LIN {X 0,Y 573.093,Z 692.429,A -85,B 0,C 180,E1 -2257.751,E2 -2257.751} C_VEL
LIN {X 0,Y 573.135,Z 684.656,A -85,B 0,C 180,E1 -2259.172,E2 -2259.172} C_VEL
LIN {X 0,Y 573.27,Z 676.378,A -85,B 0,C 180,E1 -2260.417,E2 -2260.417} C_VEL
LIN {X 0,Y 573.384,Z 666.402,A -85,B 0,C 180,E1 -2261.667,E2 -2261.667} C_VEL
LIN {X 0,Y 573.566,Z 656.201,A -85,B 0,C 180,E1 -2262.741,E2 -2262.741} C_VEL
LIN {X 0,Y 573.742,Z 644.034,A -85,B 0,C 180,E1 -2263.818,E2 -2263.818} C_VEL
LIN {X 0,Y 573.958,Z 630.922,A -85,B 0,C 180,E1 -2264.78,E2 -2264.78} C_VEL
LIN {X 0,Y 574.109,Z 618.538,A -85,B 0,C 180,E1 -2265.531,E2 -2265.531} C_VEL
LIN {X 0,Y 574.343,Z 603.86,A -85,B 0,C 180,E1 -2266.254,E2 -2266.254} C_VEL
LIN {X 0,Y 574.537,Z 589.652,A -85,B 0,C 180,E1 -2266.796,E2 -2266.796} C_VEL
LIN {X 0,Y 574.697,Z 574.641,A -85,B 0,C 180,E1 -2267.221,E2 -2267.221} C_VEL
LIN {X 0,Y 574.75,Z 559.765,A -85,B 0,C 180,E1 -2267.501,E2 -2267.501} C_VEL
LIN {X 0,Y 575.189,Z 405.134,A -85,B 0,C 180,E1 -2269.487,E2 -2269.487} C_VEL
LIN {X 0,Y 574.004,Z 398.788,A -85,B 0,C 180,E1 -2269.625,E2 -2269.625} C_VEL
LIN {X 0,Y 574.346,Z 373.403,A -85,B 0,C 180,E1 -2272.67,E2 -2272.67} C_VEL
LIN {X 0,Y 574.669,Z 351.554,A -85,B 0,C 180,E1 -2275.342,E2 -2275.342} C_VEL
LIN {X 0,Y 573.967,Z 346.839,A -85,B 0,C 180,E1 -2275.959,E2 -2275.959} C_VEL
LIN {X 0,Y 573.219,Z 343.711,A -85,B 0,C 180,E1 -2276.413,E2 -2276.413} C_VEL
LIN {X 0,Y 573.236,Z 343.702,A -85,B 0,C 180,E1 -2279.366,E2 -2279.366} C_VEL
LIN {X 0,Y 573.239,Z 343.709,A -85,B 0,C 180,E1 -2282.226,E2 -2282.226} C_VEL
LIN {X 0,Y 573.211,Z 343.705,A -85,B 0,C 180,E1 -2284.768,E2 -2284.768} C_VEL
LIN {X 0,Y 573.211,Z 343.707,A -85,B 0,C 180,E1 -2287.808,E2 -2287.808} C_VEL
LIN {X 0,Y 573.235,Z 343.704,A -85,B 0,C 180,E1 -2290.524,E2 -2290.524} C_VEL
LIN {X 0,Y 573.189,Z 343.705,A -85,B 0,C 180,E1 -2293.362,E2 -2293.362} C_VEL
LIN {X 0,Y 573.193,Z 343.712,A -85,B 0,C 180,E1 -2296.334,E2 -2296.334} C_VEL
LIN {X 0,Y 573.191,Z 343.709,A -85,B 0,C 180,E1 -2298.54,E2 -2298.54} C_VEL
LIN {X 0,Y 573.219,Z 343.701,A -85,B 0,C 180,E1 -2301.297,E2 -2301.297} C_VEL
LIN {X 0,Y 573.172,Z 343.715,A -85,B 0,C 180,E1 -2304.021,E2 -2304.021} C_VEL
LIN {X 0,Y 573.236,Z 343.703,A -85,B 0,C 180,E1 -2306.516,E2 -2306.516} C_VEL
LIN {X 0,Y 573.208,Z 343.703,A -85,B 0,C 180,E1 -2309.118,E2 -2309.118} C_VEL
LIN {X 0,Y 573.188,Z 343.713,A -85,B 0,C 180,E1 -2311.98,E2 -2311.98} C_VEL
LIN {X 0,Y 573.213,Z 343.705,A -85,B 0,C 180,E1 -2314.588,E2 -2314.588} C_VEL
LIN {X 0,Y 573.201,Z 343.707,A -85,B 0,C 180,E1 -2317.661,E2 -2317.661} C_VEL
LIN {X 0,Y 573.253,Z 343.698,A -85,B 0,C 180,E1 -2320.731,E2 -2320.731} C_VEL
LIN {X 0,Y 573.191,Z 343.708,A -85,B 0,C 180,E1 -2323.62,E2 -2323.62} C_VEL
LIN {X 0,Y 573.239,Z 343.705,A -85,B 0,C 180,E1 -2325.806,E2 -2325.806} C_VEL
LIN {X 0,Y 573.247,Z 343.699,A -85,B 0,C 180,E1 -2328.745,E2 -2328.745} C_VEL
LIN {X 0,Y 573.228,Z 343.703,A -85,B 0,C 180,E1 -2331.54,E2 -2331.54} C_VEL
LIN {X 0,Y 573.259,Z 343.701,A -85,B 0,C 180,E1 -2334.372,E2 -2334.372} C_VEL
LIN {X 0,Y 573.297,Z 343.7,A -85,B 0,C 180,E1 -2337.893,E2 -2337.893} C_VEL
LIN {X 0,Y 573.303,Z 343.701,A -85,B 0,C 180,E1 -2340,E2 -2340} C_VEL
LIN {X 0,Y 573.255,Z 343.697,A -85,B 0,C 180,E1 -2342.811,E2 -2342.811} C_VEL
LIN {X 0,Y 573.252,Z 343.702,A -85,B 0,C 180,E1 -2345.629,E2 -2345.629} C_VEL
LIN {X 0,Y 573.228,Z 343.703,A -85,B 0,C 180,E1 -2348.461,E2 -2348.461} C_VEL
LIN {X 0,Y 573.219,Z 343.703,A -85,B 0,C 180,E1 -2351.313,E2 -2351.313} C_VEL
LIN {X 0,Y 573.255,Z 343.7,A -85,B 0,C 180,E1 -2354.42,E2 -2354.42} C_VEL
LIN {X 0,Y 573.179,Z 343.707,A -85,B 0,C 180,E1 -2357.114,E2 -2357.114} C_VEL
LIN {X 0,Y 573.25,Z 343.699,A -85,B 0,C 180,E1 -2359.331,E2 -2359.331} C_VEL
LIN {X 0,Y 573.202,Z 343.707,A -85,B 0,C 180,E1 -2362.339,E2 -2362.339} C_VEL
LIN {X 0,Y 573.189,Z 343.708,A -85,B 0,C 180,E1 -2364.354,E2 -2364.354} C_VEL
LIN {X 0,Y 572.546,Z 343.788,A -85,B 0,C 180,E1 -2364.94,E2 -2364.94} C_VEL
LIN {X 0,Y 569.708,Z 344.149,A -85,B 0,C 180,E1 -2365.892,E2 -2365.892} C_VEL
LIN {X 0,Y 567.287,Z 344.447,A -85,B 0,C 180,E1 -2366.658,E2 -2366.658} C_VEL
LIN {X 0,Y 566.232,Z 344.574,A -85,B 0,C 180,E1 -2367.249,E2 -2367.249} C_VEL
LIN {X 0,Y 566.139,Z 344.585,A -85,B 0,C 180,E1 -2367.449,E2 -2367.449} C_VEL
LIN {X 0,Y 566.154,Z 344.582,A -85,B 0,C 180,E1 -2370.595,E2 -2370.595} C_VEL
LIN {X 0,Y 566.196,Z 344.577,A -85,B 0,C 180,E1 -2373.104,E2 -2373.104} C_VEL
LIN {X 0,Y 566.128,Z 344.592,A -85,B 0,C 180,E1 -2375.695,E2 -2375.695} C_VEL
LIN {X 0,Y 566.191,Z 344.578,A -85,B 0,C 180,E1 -2378.558,E2 -2378.558} C_VEL
LIN {X 0,Y 566.145,Z 344.583,A -85,B 0,C 180,E1 -2381.143,E2 -2381.143} C_VEL
LIN {X 0,Y 566.148,Z 344.589,A -85,B 0,C 180,E1 -2384.041,E2 -2384.041} C_VEL
LIN {X 0,Y 566.178,Z 344.579,A -85,B 0,C 180,E1 -2387.086,E2 -2387.086} C_VEL
LIN {X 0,Y 566.201,Z 344.578,A -85,B 0,C 180,E1 -2390.316,E2 -2390.316} C_VEL
LIN {X 0,Y 566.167,Z 344.584,A -85,B 0,C 180,E1 -2393.429,E2 -2393.429} C_VEL
LIN {X 0,Y 566.191,Z 344.58,A -85,B 0,C 180,E1 -2396.27,E2 -2396.27} C_VEL
LIN {X 0,Y 566.182,Z 344.578,A -85,B 0,C 180,E1 -2398.926,E2 -2398.926} C_VEL
LIN {X 0,Y 566.147,Z 344.591,A -85,B 0,C 180,E1 -2401.855,E2 -2401.855} C_VEL
LIN {X 0,Y 566.184,Z 344.58,A -85,B 0,C 180,E1 -2404.251,E2 -2404.251} C_VEL
LIN {X 0,Y 566.164,Z 344.58,A -85,B 0,C 180,E1 -2406.722,E2 -2406.722} C_VEL
LIN {X 0,Y 566.2,Z 344.585,A -85,B 0,C 180,E1 -2409.664,E2 -2409.664} C_VEL
LIN {X 0,Y 566.17,Z 344.586,A -85,B 0,C 180,E1 -2411.922,E2 -2411.922} C_VEL
LIN {X 0,Y 566.185,Z 344.578,A -85,B 0,C 180,E1 -2414.891,E2 -2414.891} C_VEL
LIN {X 0,Y 566.214,Z 344.582,A -85,B 0,C 180,E1 -2417.82,E2 -2417.82} C_VEL
LIN {X 0,Y 566.164,Z 344.585,A -85,B 0,C 180,E1 -2419.993,E2 -2419.993} C_VEL
LIN {X 0,Y 566.192,Z 344.58,A -85,B 0,C 180,E1 -2422.153,E2 -2422.153} C_VEL
LIN {X 0,Y 566.261,Z 344.569,A -85,B 0,C 180,E1 -2425.017,E2 -2425.017} C_VEL
LIN {X 0,Y 566.281,Z 344.572,A -85,B 0,C 180,E1 -2427.867,E2 -2427.867} C_VEL
LIN {X 0,Y 566.288,Z 344.569,A -85,B 0,C 180,E1 -2430.001,E2 -2430.001} C_VEL
LIN {X 0,Y 566.248,Z 344.57,A -85,B 0,C 180,E1 -2432.847,E2 -2432.847} C_VEL
LIN {X 0,Y 566.247,Z 344.579,A -85,B 0,C 180,E1 -2435.699,E2 -2435.699} C_VEL
LIN {X 0,Y 566.201,Z 344.576,A -85,B 0,C 180,E1 -2438.567,E2 -2438.567} C_VEL
LIN {X 0,Y 566.245,Z 344.578,A -85,B 0,C 180,E1 -2441.455,E2 -2441.455} C_VEL
LIN {X 0,Y 566.224,Z 344.573,A -85,B 0,C 180,E1 -2444.501,E2 -2444.501} C_VEL
LIN {X 0,Y 566.159,Z 344.587,A -85,B 0,C 180,E1 -2447.334,E2 -2447.334} C_VEL
LIN {X 0,Y 566.205,Z 344.586,A -85,B 0,C 180,E1 -2449.582,E2 -2449.582} C_VEL
LIN {X 0,Y 566.191,Z 344.582,A -85,B 0,C 180,E1 -2451.864,E2 -2451.864} C_VEL
LIN {X 0,Y 566.185,Z 344.58,A -85,B 0,C 180,E1 -2455.022,E2 -2455.022} C_VEL
LIN {X 0,Y 566.172,Z 344.586,A -85,B 0,C 180,E1 -2457.342,E2 -2457.342} C_VEL
LIN {X 0,Y 566.177,Z 344.585,A -85,B 0,C 180,E1 -2459.771,E2 -2459.771} C_VEL
LIN {X 0,Y 566.205,Z 344.575,A -85,B 0,C 180,E1 -2462.429,E2 -2462.429} C_VEL
LIN {X 0,Y 566.174,Z 344.581,A -85,B 0,C 180,E1 -2464.988,E2 -2464.988} C_VEL
LIN {X 0,Y 566.197,Z 344.587,A -85,B 0,C 180,E1 -2467.462,E2 -2467.462} C_VEL
LIN {X 0,Y 566.212,Z 344.577,A -85,B 0,C 180,E1 -2470.199,E2 -2470.199} C_VEL
LIN {X 0,Y 566.197,Z 344.581,A -85,B 0,C 180,E1 -2473.055,E2 -2473.055} C_VEL
LIN {X 0,Y 566.164,Z 344.587,A -85,B 0,C 180,E1 -2476.053,E2 -2476.053} C_VEL
LIN {X 0,Y 566.24,Z 344.709,A -85,B 0,C 180,E1 -2477.589,E2 -2477.589} C_VEL
LIN {X 0,Y 567.165,Z 350.607,A -85,B 0,C 180,E1 -2478.475,E2 -2478.475} C_VEL
LIN {X 0,Y 566.907,Z 369.86,A -85,B 0,C 180,E1 -2481.181,E2 -2481.181} C_VEL
LIN {X 0,Y 568.471,Z 377.974,A -85,B 0,C 180,E1 -2481.356,E2 -2481.356} C_VEL
LIN {X 0,Y 567.987,Z 535.046,A -85,B 0,C 180,E1 -2483.412,E2 -2483.412} C_VEL
LIN {X 0,Y 567.798,Z 550.912,A -85,B 0,C 180,E1 -2483.769,E2 -2483.769} C_VEL
LIN {X 0,Y 567.621,Z 565.523,A -85,B 0,C 180,E1 -2484.25,E2 -2484.25} C_VEL
LIN {X 0,Y 567.413,Z 579.054,A -85,B 0,C 180,E1 -2484.834,E2 -2484.834} C_VEL
LIN {X 0,Y 567.18,Z 590.968,A -85,B 0,C 180,E1 -2485.466,E2 -2485.466} C_VEL
LIN {X 0,Y 566.958,Z 603.145,A -85,B 0,C 180,E1 -2486.234,E2 -2486.234} C_VEL
LIN {X 0,Y 566.694,Z 616.436,A -85,B 0,C 180,E1 -2487.254,E2 -2487.254} C_VEL
LIN {X 0,Y 566.474,Z 628.594,A -85,B 0,C 180,E1 -2488.387,E2 -2488.387} C_VEL
LIN {X 0,Y 566.315,Z 639.636,A -85,B 0,C 180,E1 -2489.621,E2 -2489.621} C_VEL
LIN {X 0,Y 566.174,Z 648.775,A -85,B 0,C 180,E1 -2490.842,E2 -2490.842} C_VEL
LIN {X 0,Y 566.081,Z 656.346,A -85,B 0,C 180,E1 -2492.051,E2 -2492.051} C_VEL
LIN {X 0,Y 565.985,Z 663.625,A -85,B 0,C 180,E1 -2493.447,E2 -2493.447} C_VEL
LIN {X 0,Y 565.937,Z 668.628,A -85,B 0,C 180,E1 -2494.632,E2 -2494.632} C_VEL
LIN {X 0,Y 565.902,Z 672.635,A -85,B 0,C 180,E1 -2495.806,E2 -2495.806} C_VEL
LIN {X 0,Y 565.858,Z 676.627,A -85,B 0,C 180,E1 -2497.355,E2 -2497.355} C_VEL
LIN {X 0,Y 565.879,Z 679.184,A -85,B 0,C 180,E1 -2498.889,E2 -2498.889} C_VEL
LIN {X 0,Y 565.828,Z 680.353,A -85,B 0,C 180,E1 -2500.405,E2 -2500.405} C_VEL
LIN {X 0,Y 565.834,Z 680.288,A -85,B 0,C 180,E1 -2501.909,E2 -2501.909} C_VEL
LIN {X 0,Y 565.849,Z 678.914,A -85,B 0,C 180,E1 -2503.401,E2 -2503.401} C_VEL
LIN {X 0,Y 565.836,Z 676.338,A -85,B 0,C 180,E1 -2504.88,E2 -2504.88} C_VEL
LIN {X 0,Y 565.906,Z 672.428,A -85,B 0,C 180,E1 -2506.351,E2 -2506.351} C_VEL
LIN {X 0,Y 565.95,Z 667.235,A -85,B 0,C 180,E1 -2507.813,E2 -2507.813} C_VEL
LIN {X 0,Y 566.022,Z 660.559,A -85,B 0,C 180,E1 -2509.266,E2 -2509.266} C_VEL
LIN {X 0,Y 566.104,Z 652.29,A -85,B 0,C 180,E1 -2510.712,E2 -2510.712} C_VEL
LIN {X 0,Y 566.277,Z 643.544,A -85,B 0,C 180,E1 -2511.974,E2 -2511.974} C_VEL
LIN {X 0,Y 566.387,Z 633.439,A -85,B 0,C 180,E1 -2513.188,E2 -2513.188} C_VEL
LIN {X 0,Y 566.619,Z 622.414,A -85,B 0,C 180,E1 -2514.305,E2 -2514.305} C_VEL
LIN {X 0,Y 566.811,Z 610.787,A -85,B 0,C 180,E1 -2515.288,E2 -2515.288} C_VEL
LIN {X 0,Y 567.057,Z 598.317,A -85,B 0,C 180,E1 -2516.18,E2 -2516.18} C_VEL
LIN {X 0,Y 567.321,Z 584.602,A -85,B 0,C 180,E1 -2516.982,E2 -2516.982} C_VEL
LIN {X 0,Y 567.525,Z 570.387,A -85,B 0,C 180,E1 -2517.649,E2 -2517.649} C_VEL
LIN {X 0,Y 567.743,Z 555.438,A -85,B 0,C 180,E1 -2518.182,E2 -2518.182} C_VEL
LIN {X 0,Y 567.943,Z 540.077,A -85,B 0,C 180,E1 -2518.582,E2 -2518.582} C_VEL
LIN {X 0,Y 568.037,Z 521.708,A -85,B 0,C 180,E1 -2518.87,E2 -2518.87} C_VEL
LIN {X 0,Y 568.361,Z 376.894,A -85,B 0,C 180,E1 -2520.753,E2 -2520.753} C_VEL
LIN {X 0,Y 566.902,Z 369.852,A -85,B 0,C 180,E1 -2520.91,E2 -2520.91} C_VEL
LIN {X 0,Y 567.185,Z 351.045,A -85,B 0,C 180,E1 -2523.552,E2 -2523.552} C_VEL
LIN {X 0,Y 566.799,Z 347.4,A -85,B 0,C 180,E1 -2524.088,E2 -2524.088} C_VEL
LIN {X 0,Y 566.205,Z 344.584,A -85,B 0,C 180,E1 -2524.538,E2 -2524.538} C_VEL
LIN {X 0,Y 566.244,Z 344.575,A -85,B 0,C 180,E1 -2527.13,E2 -2527.13} C_VEL
LIN {X 0,Y 566.173,Z 344.584,A -85,B 0,C 180,E1 -2530.008,E2 -2530.008} C_VEL
LIN {X 0,Y 566.235,Z 344.578,A -85,B 0,C 180,E1 -2532.181,E2 -2532.181} C_VEL
LIN {X 0,Y 566.196,Z 344.579,A -85,B 0,C 180,E1 -2535.109,E2 -2535.109} C_VEL
LIN {X 0,Y 566.191,Z 344.579,A -85,B 0,C 180,E1 -2537.332,E2 -2537.332} C_VEL
LIN {X 0,Y 566.203,Z 344.577,A -85,B 0,C 180,E1 -2539.581,E2 -2539.581} C_VEL
LIN {X 0,Y 566.193,Z 344.58,A -85,B 0,C 180,E1 -2541.862,E2 -2541.862} C_VEL
LIN {X 0,Y 566.182,Z 344.58,A -85,B 0,C 180,E1 -2545.021,E2 -2545.021} C_VEL
LIN {X 0,Y 566.163,Z 344.582,A -85,B 0,C 180,E1 -2547.341,E2 -2547.341} C_VEL
LIN {X 0,Y 566.161,Z 344.585,A -85,B 0,C 180,E1 -2549.771,E2 -2549.771} C_VEL
LIN {X 0,Y 566.181,Z 344.585,A -85,B 0,C 180,E1 -2552.425,E2 -2552.425} C_VEL
LIN {X 0,Y 566.162,Z 344.582,A -85,B 0,C 180,E1 -2554.986,E2 -2554.986} C_VEL
LIN {X 0,Y 566.182,Z 344.58,A -85,B 0,C 180,E1 -2557.462,E2 -2557.462} C_VEL
LIN {X 0,Y 566.179,Z 344.587,A -85,B 0,C 180,E1 -2560.201,E2 -2560.201} C_VEL
LIN {X 0,Y 566.142,Z 344.584,A -85,B 0,C 180,E1 -2563.06,E2 -2563.06} C_VEL
LIN {X 0,Y 566.143,Z 344.592,A -85,B 0,C 180,E1 -2566.054,E2 -2566.054} C_VEL
LIN {X 0,Y 566.133,Z 344.585,A -85,B 0,C 180,E1 -2568.856,E2 -2568.856} C_VEL
LIN {X 0,Y 566.161,Z 344.587,A -85,B 0,C 180,E1 -2571.634,E2 -2571.634} C_VEL
LIN {X 0,Y 566.135,Z 344.59,A -85,B 0,C 180,E1 -2574.305,E2 -2574.305} C_VEL
LIN {X 0,Y 566.164,Z 344.583,A -85,B 0,C 180,E1 -2576.893,E2 -2576.893} C_VEL
LIN {X 0,Y 566.162,Z 344.588,A -85,B 0,C 180,E1 -2579.405,E2 -2579.405} C_VEL
LIN {X 0,Y 566.144,Z 344.593,A -85,B 0,C 180,E1 -2581.853,E2 -2581.853} C_VEL
LIN {X 0,Y 566.16,Z 344.667,A -85,B 0,C 180,E1 -2583.425,E2 -2583.425} C_VEL
LIN {X 0,Y 567.712,Z 351.329,A -85,B 0,C 180,E1 -2584.323,E2 -2584.323} C_VEL
LIN {X 0,Y 567.602,Z 368.07,A -85,B 0,C 180,E1 -2586.385,E2 -2586.385} C_VEL
LIN {X 0,Y 567.272,Z 388.991,A -85,B 0,C 180,E1 -2588.943,E2 -2588.943} C_VEL
LIN {X 0,Y 567.118,Z 398.912,A -85,B 0,C 180,E1 -2590.141,E2 -2590.141} C_VEL
LIN {X 0,Y 568.525,Z 407.122,A -85,B 0,C 180,E1 -2590.301,E2 -2590.301} C_VEL
LIN {X 0,Y 567.986,Z 564.907,A -85,B 0,C 180,E1 -2592.363,E2 -2592.363} C_VEL
LIN {X 0,Y 567.835,Z 580.673,A -85,B 0,C 180,E1 -2592.719,E2 -2592.719} C_VEL
LIN {X 0,Y 567.628,Z 596.017,A -85,B 0,C 180,E1 -2593.223,E2 -2593.223} C_VEL
LIN {X 0,Y 567.444,Z 609.753,A -85,B 0,C 180,E1 -2593.818,E2 -2593.818} C_VEL
LIN {X 0,Y 567.153,Z 623.23,A -85,B 0,C 180,E1 -2594.548,E2 -2594.548} C_VEL
LIN {X 0,Y 566.934,Z 635.507,A -85,B 0,C 180,E1 -2595.358,E2 -2595.358} C_VEL
LIN {X 0,Y 566.672,Z 648.28,A -85,B 0,C 180,E1 -2596.37,E2 -2596.37} C_VEL
LIN {X 0,Y 566.492,Z 659.74,A -85,B 0,C 180,E1 -2597.46,E2 -2597.46} C_VEL
LIN {X 0,Y 566.27,Z 670.305,A -85,B 0,C 180,E1 -2598.658,E2 -2598.658} C_VEL
LIN {X 0,Y 566.209,Z 678.85,A -85,B 0,C 180,E1 -2599.811,E2 -2599.811} C_VEL
LIN {X 0,Y 566.057,Z 686.729,A -85,B 0,C 180,E1 -2601.071,E2 -2601.071} C_VEL
LIN {X 0,Y 565.998,Z 694.085,A -85,B 0,C 180,E1 -2602.508,E2 -2602.508} C_VEL
LIN {X 0,Y 565.958,Z 699.919,A -85,B 0,C 180,E1 -2603.94,E2 -2603.94} C_VEL
LIN {X 0,Y 565.867,Z 703.383,A -85,B 0,C 180,E1 -2605.011,E2 -2605.011} C_VEL
LIN {X 0,Y 565.91,Z 706.888,A -85,B 0,C 180,E1 -2606.439,E2 -2606.439} C_VEL
LIN {X 0,Y 565.839,Z 709.191,A -85,B 0,C 180,E1 -2607.864,E2 -2607.864} C_VEL
LIN {X 0,Y 565.837,Z 710.349,A -85,B 0,C 180,E1 -2609.287,E2 -2609.287} C_VEL
LIN {X 0,Y 565.836,Z 710.349,A -85,B 0,C 180,E1 -2610.711,E2 -2610.711} C_VEL
LIN {X 0,Y 565.838,Z 709.191,A -85,B 0,C 180,E1 -2612.134,E2 -2612.134} C_VEL
LIN {X 0,Y 565.91,Z 706.889,A -85,B 0,C 180,E1 -2613.559,E2 -2613.559} C_VEL
LIN {X 0,Y 565.866,Z 703.389,A -85,B 0,C 180,E1 -2614.986,E2 -2614.986} C_VEL
LIN {X 0,Y 565.941,Z 698.613,A -85,B 0,C 180,E1 -2616.416,E2 -2616.416} C_VEL
LIN {X 0,Y 566.013,Z 692.428,A -85,B 0,C 180,E1 -2617.849,E2 -2617.849} C_VEL
LIN {X 0,Y 566.07,Z 684.655,A -85,B 0,C 180,E1 -2619.287,E2 -2619.287} C_VEL
LIN {X 0,Y 566.238,Z 676.377,A -85,B 0,C 180,E1 -2620.548,E2 -2620.548} C_VEL
LIN {X 0,Y 566.365,Z 666.402,A -85,B 0,C 180,E1 -2621.814,E2 -2621.814} C_VEL
LIN {X 0,Y 566.584,Z 656.2,A -85,B 0,C 180,E1 -2622.9,E2 -2622.9} C_VEL
LIN {X 0,Y 566.798,Z 644.034,A -85,B 0,C 180,E1 -2623.991,E2 -2623.991} C_VEL
LIN {X 0,Y 567.037,Z 631.358,A -85,B 0,C 180,E1 -2624.935,E2 -2624.935} C_VEL
LIN {X 0,Y 567.228,Z 618.535,A -85,B 0,C 180,E1 -2625.724,E2 -2625.724} C_VEL
LIN {X 0,Y 567.479,Z 603.857,A -85,B 0,C 180,E1 -2626.456,E2 -2626.456} C_VEL
LIN {X 0,Y 567.74,Z 589.651,A -85,B 0,C 180,E1 -2627.003,E2 -2627.003} C_VEL
LIN {X 0,Y 567.919,Z 575.293,A -85,B 0,C 180,E1 -2627.416,E2 -2627.416} C_VEL
LIN {X 0,Y 567.981,Z 560.881,A -85,B 0,C 180,E1 -2627.699,E2 -2627.699} C_VEL
LIN {X 0,Y 568.463,Z 405.776,A -85,B 0,C 180,E1 -2629.719,E2 -2629.719} C_VEL
LIN {X 0,Y 567.132,Z 398.845,A -85,B 0,C 180,E1 -2629.866,E2 -2629.866} C_VEL
LIN {X 0,Y 567.489,Z 374.964,A -85,B 0,C 180,E1 -2632.767,E2 -2632.767} C_VEL
LIN {X 0,Y 567.842,Z 353.148,A -85,B 0,C 180,E1 -2635.455,E2 -2635.455} C_VEL
LIN {X 0,Y 567.076,Z 348.267,A -85,B 0,C 180,E1 -2636.1,E2 -2636.1} C_VEL
LIN {X 0,Y 566.158,Z 344.59,A -85,B 0,C 180,E1 -2636.617,E2 -2636.617} C_VEL
LIN {X 0,Y 566.166,Z 344.584,A -85,B 0,C 180,E1 -2638.953,E2 -2638.953} C_VEL
LIN {X 0,Y 566.182,Z 344.58,A -85,B 0,C 180,E1 -2641.421,E2 -2641.421} C_VEL
LIN {X 0,Y 566.189,Z 344.584,A -85,B 0,C 180,E1 -2643.956,E2 -2643.956} C_VEL
LIN {X 0,Y 566.164,Z 344.585,A -85,B 0,C 180,E1 -2646.571,E2 -2646.571} C_VEL
LIN {X 0,Y 566.199,Z 344.579,A -85,B 0,C 180,E1 -2649.684,E2 -2649.684} C_VEL
LIN {X 0,Y 566.176,Z 344.579,A -85,B 0,C 180,E1 -2652.915,E2 -2652.915} C_VEL
LIN {X 0,Y 566.144,Z 344.591,A -85,B 0,C 180,E1 -2656.052,E2 -2656.052} C_VEL
LIN {X 0,Y 566.144,Z 344.584,A -85,B 0,C 180,E1 -2658.858,E2 -2658.858} C_VEL
LIN {X 0,Y 566.189,Z 344.578,A -85,B 0,C 180,E1 -2661.442,E2 -2661.442} C_VEL
LIN {X 0,Y 566.127,Z 344.592,A -85,B 0,C 180,E1 -2664.305,E2 -2664.305} C_VEL
LIN {X 0,Y 566.194,Z 344.577,A -85,B 0,C 180,E1 -2666.896,E2 -2666.896} C_VEL
LIN {X 0,Y 566.157,Z 344.582,A -85,B 0,C 180,E1 -2669.406,E2 -2669.406} C_VEL
LIN {X 0,Y 566.134,Z 344.59,A -85,B 0,C 180,E1 -2671.853,E2 -2671.853} C_VEL
LIN {X 0,Y 566.173,Z 344.587,A -85,B 0,C 180,E1 -2674.249,E2 -2674.249} C_VEL
LIN {X 0,Y 566.15,Z 344.583,A -85,B 0,C 180,E1 -2676.72,E2 -2676.72} C_VEL
LIN {X 0,Y 566.177,Z 344.582,A -85,B 0,C 180,E1 -2679.662,E2 -2679.662} C_VEL
LIN {X 0,Y 566.155,Z 344.589,A -85,B 0,C 180,E1 -2681.921,E2 -2681.921} C_VEL
LIN {X 0,Y 566.168,Z 344.58,A -85,B 0,C 180,E1 -2684.89,E2 -2684.89} C_VEL
LIN {X 0,Y 566.164,Z 344.586,A -85,B 0,C 180,E1 -2687.818,E2 -2687.818} C_VEL
LIN {X 0,Y 566.149,Z 344.592,A -85,B 0,C 180,E1 -2689.992,E2 -2689.992} C_VEL
LIN {X 0,Y 566.173,Z 344.587,A -85,B 0,C 180,E1 -2692.152,E2 -2692.152} C_VEL
LIN {X 0,Y 566.237,Z 344.571,A -85,B 0,C 180,E1 -2695.016,E2 -2695.016} C_VEL
LIN {X 0,Y 566.267,Z 344.575,A -85,B 0,C 180,E1 -2697.866,E2 -2697.866} C_VEL
LIN {X 0,Y 566.271,Z 344.577,A -85,B 0,C 180,E1 -2700,E2 -2700} C_VEL
LIN {X 0,Y 566.223,Z 344.573,A -85,B 0,C 180,E1 -2702.846,E2 -2702.846} C_VEL
LIN {X 0,Y 566.222,Z 344.578,A -85,B 0,C 180,E1 -2705.699,E2 -2705.699} C_VEL
LIN {X 0,Y 566.178,Z 344.58,A -85,B 0,C 180,E1 -2708.567,E2 -2708.567} C_VEL
LIN {X 0,Y 566.177,Z 344.581,A -85,B 0,C 180,E1 -2711.456,E2 -2711.456} C_VEL
LIN {X 0,Y 566.209,Z 344.577,A -85,B 0,C 180,E1 -2714.503,E2 -2714.503} C_VEL
LIN {X 0,Y 566.145,Z 344.584,A -85,B 0,C 180,E1 -2717.334,E2 -2717.334} C_VEL
LIN {X 0,Y 566.183,Z 344.582,A -85,B 0,C 180,E1 -2719.582,E2 -2719.582} C_VEL
LIN {X 0,Y 566.167,Z 344.589,A -85,B 0,C 180,E1 -2721.864,E2 -2721.864} C_VEL
LIN {X 0,Y 566.139,Z 344.587,A -85,B 0,C 180,E1 -2724.351,E2 -2724.351} C_VEL
LIN {X 0,Y 566.154,Z 344.582,A -85,B 0,C 180,E1 -2726.652,E2 -2726.652} C_VEL
LIN {X 0,Y 566.139,Z 344.585,A -85,B 0,C 180,E1 -2727.449,E2 -2727.449} C_VEL
LIN {X 0,Y 565.453,Z 344.677,A -85,B 0,C 180,E1 -2728.043,E2 -2728.043} C_VEL
LIN {X 0,Y 562.598,Z 345.028,A -85,B 0,C 180,E1 -2729.007,E2 -2729.007} C_VEL
LIN {X 0,Y 560.205,Z 345.331,A -85,B 0,C 180,E1 -2729.782,E2 -2729.782} C_VEL
LIN {X 0,Y 559.189,Z 345.452,A -85,B 0,C 180,E1 -2730.381,E2 -2730.381} C_VEL
LIN {X 0,Y 559.112,Z 345.46,A -85,B 0,C 180,E1 -2730.584,E2 -2730.584} C_VEL
LIN {X 0,Y 559.14,Z 345.455,A -85,B 0,C 180,E1 -2732.717,E2 -2732.717} C_VEL
LIN {X 0,Y 559.104,Z 345.462,A -85,B 0,C 180,E1 -2735.326,E2 -2735.326} C_VEL
LIN {X 0,Y 559.113,Z 345.466,A -85,B 0,C 180,E1 -2738.02,E2 -2738.02} C_VEL
LIN {X 0,Y 559.147,Z 345.463,A -85,B 0,C 180,E1 -2739.942,E2 -2739.942} C_VEL
LIN {X 0,Y 559.129,Z 345.457,A -85,B 0,C 180,E1 -2742.747,E2 -2742.747} C_VEL
LIN {X 0,Y 559.114,Z 345.468,A -85,B 0,C 180,E1 -2745.765,E2 -2745.765} C_VEL
LIN {X 0,Y 559.116,Z 345.462,A -85,B 0,C 180,E1 -2748.227,E2 -2748.227} C_VEL
LIN {X 0,Y 559.161,Z 345.454,A -85,B 0,C 180,E1 -2751.194,E2 -2751.194} C_VEL
LIN {X 0,Y 559.108,Z 345.47,A -85,B 0,C 180,E1 -2753.789,E2 -2753.789} C_VEL
LIN {X 0,Y 559.141,Z 345.456,A -85,B 0,C 180,E1 -2756.425,E2 -2756.425} C_VEL
LIN {X 0,Y 559.147,Z 345.455,A -85,B 0,C 180,E1 -2758.982,E2 -2758.982} C_VEL
LIN {X 0,Y 559.105,Z 345.467,A -85,B 0,C 180,E1 -2761.632,E2 -2761.632} C_VEL
LIN {X 0,Y 559.15,Z 345.462,A -85,B 0,C 180,E1 -2763.903,E2 -2763.903} C_VEL
LIN {X 0,Y 559.132,Z 345.456,A -85,B 0,C 180,E1 -2766.574,E2 -2766.574} C_VEL
LIN {X 0,Y 559.171,Z 345.456,A -85,B 0,C 180,E1 -2769.397,E2 -2769.397} C_VEL
LIN {X 0,Y 559.121,Z 345.467,A -85,B 0,C 180,E1 -2771.686,E2 -2771.686} C_VEL
LIN {X 0,Y 559.136,Z 345.462,A -85,B 0,C 180,E1 -2773.948,E2 -2773.948} C_VEL
LIN {X 0,Y 559.157,Z 345.456,A -85,B 0,C 180,E1 -2776.185,E2 -2776.185} C_VEL
LIN {X 0,Y 559.192,Z 345.451,A -85,B 0,C 180,E1 -2779.135,E2 -2779.135} C_VEL
LIN {X 0,Y 559.145,Z 345.459,A -85,B 0,C 180,E1 -2782.054,E2 -2782.054} C_VEL
LIN {X 0,Y 559.236,Z 345.444,A -85,B 0,C 180,E1 -2784.954,E2 -2784.954} C_VEL
LIN {X 0,Y 559.252,Z 345.448,A -85,B 0,C 180,E1 -2787.841,E2 -2787.841} C_VEL
LIN {X 0,Y 559.257,Z 345.445,A -85,B 0,C 180,E1 -2790.001,E2 -2790.001} C_VEL
LIN {X 0,Y 559.216,Z 345.446,A -85,B 0,C 180,E1 -2792.883,E2 -2792.883} C_VEL
LIN {X 0,Y 559.216,Z 345.453,A -85,B 0,C 180,E1 -2795.771,E2 -2795.771} C_VEL
LIN {X 0,Y 559.166,Z 345.452,A -85,B 0,C 180,E1 -2798.676,E2 -2798.676} C_VEL
LIN {X 0,Y 559.203,Z 345.458,A -85,B 0,C 180,E1 -2801.601,E2 -2801.601} C_VEL
LIN {X 0,Y 559.187,Z 345.449,A -85,B 0,C 180,E1 -2804.588,E2 -2804.588} C_VEL
LIN {X 0,Y 559.117,Z 345.468,A -85,B 0,C 180,E1 -2807.559,E2 -2807.559} C_VEL
LIN {X 0,Y 559.168,Z 345.457,A -85,B 0,C 180,E1 -2809.838,E2 -2809.838} C_VEL
LIN {X 0,Y 559.137,Z 345.457,A -85,B 0,C 180,E1 -2812.154,E2 -2812.154} C_VEL
LIN {X 0,Y 559.145,Z 345.459,A -85,B 0,C 180,E1 -2815.178,E2 -2815.178} C_VEL
LIN {X 0,Y 559.123,Z 345.465,A -85,B 0,C 180,E1 -2817.716,E2 -2817.716} C_VEL
LIN {X 0,Y 559.142,Z 345.456,A -85,B 0,C 180,E1 -2820.184,E2 -2820.184} C_VEL
LIN {X 0,Y 559.16,Z 345.453,A -85,B 0,C 180,E1 -2822.716,E2 -2822.716} C_VEL
LIN {X 0,Y 559.123,Z 345.464,A -85,B 0,C 180,E1 -2825.325,E2 -2825.325} C_VEL
LIN {X 0,Y 559.133,Z 345.46,A -85,B 0,C 180,E1 -2828.018,E2 -2828.018} C_VEL
LIN {X 0,Y 559.16,Z 345.455,A -85,B 0,C 180,E1 -2830.813,E2 -2830.813} C_VEL
LIN {X 0,Y 559.128,Z 345.465,A -85,B 0,C 180,E1 -2833.736,E2 -2833.736} C_VEL
LIN {X 0,Y 559.116,Z 345.464,A -85,B 0,C 180,E1 -2836.263,E2 -2836.263} C_VEL
LIN {X 0,Y 559.164,Z 345.464,A -85,B 0,C 180,E1 -2837.363,E2 -2837.363} C_VEL
LIN {X 0,Y 560.276,Z 351.712,A -85,B 0,C 180,E1 -2838.331,E2 -2838.331} C_VEL
LIN {X 0,Y 559.995,Z 369.911,A -85,B 0,C 180,E1 -2840.933,E2 -2840.933} C_VEL
LIN {X 0,Y 561.801,Z 379.493,A -85,B 0,C 180,E1 -2841.132,E2 -2841.132} C_VEL
LIN {X 0,Y 561.222,Z 535.023,A -85,B 0,C 180,E1 -2843.192,E2 -2843.192} C_VEL
LIN {X 0,Y 561.025,Z 551.154,A -85,B 0,C 180,E1 -2843.561,E2 -2843.561} C_VEL
LIN {X 0,Y 560.808,Z 566.044,A -85,B 0,C 180,E1 -2844.06,E2 -2844.06} C_VEL
LIN {X 0,Y 560.566,Z 578.048,A -85,B 0,C 180,E1 -2844.581,E2 -2844.581} C_VEL
LIN {X 0,Y 560.32,Z 589.793,A -85,B 0,C 180,E1 -2845.201,E2 -2845.201} C_VEL
LIN {X 0,Y 560.058,Z 602.451,A -85,B 0,C 180,E1 -2845.996,E2 -2845.996} C_VEL
LIN {X 0,Y 559.769,Z 616.048,A -85,B 0,C 180,E1 -2847.045,E2 -2847.045} C_VEL
LIN {X 0,Y 559.517,Z 627.927,A -85,B 0,C 180,E1 -2848.159,E2 -2848.159} C_VEL
LIN {X 0,Y 559.315,Z 639.102,A -85,B 0,C 180,E1 -2849.409,E2 -2849.409} C_VEL
LIN {X 0,Y 559.133,Z 648.327,A -85,B 0,C 180,E1 -2850.645,E2 -2850.645} C_VEL
LIN {X 0,Y 559.006,Z 656.463,A -85,B 0,C 180,E1 -2851.958,E2 -2851.958} C_VEL
LIN {X 0,Y 558.92,Z 663.037,A -85,B 0,C 180,E1 -2853.225,E2 -2853.225} C_VEL
LIN {X 0,Y 558.857,Z 669.118,A -85,B 0,C 180,E1 -2854.686,E2 -2854.686} C_VEL
LIN {X 0,Y 558.819,Z 674.172,A -85,B 0,C 180,E1 -2856.268,E2 -2856.268} C_VEL
LIN {X 0,Y 558.75,Z 677.635,A -85,B 0,C 180,E1 -2857.831,E2 -2857.831} C_VEL
LIN {X 0,Y 558.739,Z 679.714,A -85,B 0,C 180,E1 -2859.378,E2 -2859.378} C_VEL
LIN {X 0,Y 558.779,Z 680.477,A -85,B 0,C 180,E1 -2860.912,E2 -2860.912} C_VEL
LIN {X 0,Y 558.747,Z 679.945,A -85,B 0,C 180,E1 -2862.429,E2 -2862.429} C_VEL
LIN {X 0,Y 558.74,Z 678.194,A -85,B 0,C 180,E1 -2863.935,E2 -2863.935} C_VEL
LIN {X 0,Y 558.784,Z 674.79,A -85,B 0,C 180,E1 -2865.571,E2 -2865.571} C_VEL
LIN {X 0,Y 558.818,Z 670.852,A -85,B 0,C 180,E1 -2866.916,E2 -2866.916} C_VEL
LIN {X 0,Y 558.867,Z 665.159,A -85,B 0,C 180,E1 -2868.392,E2 -2868.392} C_VEL
LIN {X 0,Y 558.977,Z 657.973,A -85,B 0,C 180,E1 -2869.862,E2 -2869.862} C_VEL
LIN {X 0,Y 559.117,Z 650.35,A -85,B 0,C 180,E1 -2871.142,E2 -2871.142} C_VEL
LIN {X 0,Y 559.261,Z 641.186,A -85,B 0,C 180,E1 -2872.418,E2 -2872.418} C_VEL
LIN {X 0,Y 559.404,Z 631.979,A -85,B 0,C 180,E1 -2873.507,E2 -2873.507} C_VEL
LIN {X 0,Y 559.679,Z 621.063,A -85,B 0,C 180,E1 -2874.596,E2 -2874.596} C_VEL
LIN {X 0,Y 559.855,Z 610.39,A -85,B 0,C 180,E1 -2875.5,E2 -2875.5} C_VEL
LIN {X 0,Y 560.171,Z 597.829,A -85,B 0,C 180,E1 -2876.403,E2 -2876.403} C_VEL
LIN {X 0,Y 560.483,Z 583.977,A -85,B 0,C 180,E1 -2877.215,E2 -2877.215} C_VEL
LIN {X 0,Y 560.77,Z 569.554,A -85,B 0,C 180,E1 -2877.89,E2 -2877.89} C_VEL
LIN {X 0,Y 560.948,Z 554.403,A -85,B 0,C 180,E1 -2878.429,E2 -2878.429} C_VEL
LIN {X 0,Y 561.202,Z 539.51,A -85,B 0,C 180,E1 -2878.811,E2 -2878.811} C_VEL
LIN {X 0,Y 561.295,Z 520.826,A -85,B 0,C 180,E1 -2879.103,E2 -2879.103} C_VEL
LIN {X 0,Y 561.719,Z 378.149,A -85,B 0,C 180,E1 -2880.979,E2 -2880.979} C_VEL
LIN {X 0,Y 559.99,Z 369.822,A -85,B 0,C 180,E1 -2881.17,E2 -2881.17} C_VEL
LIN {X 0,Y 560.293,Z 351.642,A -85,B 0,C 180,E1 -2883.776,E2 -2883.776} C_VEL
LIN {X 0,Y 559.2,Z 345.457,A -85,B 0,C 180,E1 -2884.776,E2 -2884.776} C_VEL
LIN {X 0,Y 559.207,Z 345.452,A -85,B 0,C 180,E1 -2887.22,E2 -2887.22} C_VEL
LIN {X 0,Y 559.134,Z 345.463,A -85,B 0,C 180,E1 -2890.135,E2 -2890.135} C_VEL
LIN {X 0,Y 559.189,Z 345.458,A -85,B 0,C 180,E1 -2892.337,E2 -2892.337} C_VEL
LIN {X 0,Y 559.144,Z 345.457,A -85,B 0,C 180,E1 -2895.305,E2 -2895.305} C_VEL
LIN {X 0,Y 559.136,Z 345.458,A -85,B 0,C 180,E1 -2897.557,E2 -2897.557} C_VEL
LIN {X 0,Y 559.167,Z 345.455,A -85,B 0,C 180,E1 -2899.837,E2 -2899.837} C_VEL
LIN {X 0,Y 559.141,Z 345.463,A -85,B 0,C 180,E1 -2902.153,E2 -2902.153} C_VEL
LIN {X 0,Y 559.141,Z 345.456,A -85,B 0,C 180,E1 -2905.177,E2 -2905.177} C_VEL
LIN {X 0,Y 559.107,Z 345.463,A -85,B 0,C 180,E1 -2907.716,E2 -2907.716} C_VEL
LIN {X 0,Y 559.133,Z 345.466,A -85,B 0,C 180,E1 -2910.184,E2 -2910.184} C_VEL
LIN {X 0,Y 559.138,Z 345.459,A -85,B 0,C 180,E1 -2912.716,E2 -2912.716} C_VEL
LIN {X 0,Y 559.115,Z 345.46,A -85,B 0,C 180,E1 -2915.325,E2 -2915.325} C_VEL
LIN {X 0,Y 559.122,Z 345.466,A -85,B 0,C 180,E1 -2918.018,E2 -2918.018} C_VEL
LIN {X 0,Y 559.133,Z 345.464,A -85,B 0,C 180,E1 -2919.937,E2 -2919.937} C_VEL
LIN {X 0,Y 559.11,Z 345.461,A -85,B 0,C 180,E1 -2922.748,E2 -2922.748} C_VEL
LIN {X 0,Y 559.113,Z 345.465,A -85,B 0,C 180,E1 -2925.765,E2 -2925.765} C_VEL
LIN {X 0,Y 559.093,Z 345.468,A -85,B 0,C 180,E1 -2928.222,E2 -2928.222} C_VEL
LIN {X 0,Y 559.137,Z 345.458,A -85,B 0,C 180,E1 -2931.196,E2 -2931.196} C_VEL
LIN {X 0,Y 559.108,Z 345.469,A -85,B 0,C 180,E1 -2933.786,E2 -2933.786} C_VEL
LIN {X 0,Y 559.125,Z 345.463,A -85,B 0,C 180,E1 -2936.422,E2 -2936.422} C_VEL
LIN {X 0,Y 559.141,Z 345.46,A -85,B 0,C 180,E1 -2938.979,E2 -2938.979} C_VEL
LIN {X 0,Y 559.105,Z 345.47,A -85,B 0,C 180,E1 -2941.631,E2 -2941.631} C_VEL
LIN {X 0,Y 559.137,Z 345.576,A -85,B 0,C 180,E1 -2943.212,E2 -2943.212} C_VEL
LIN {X 0,Y 560.909,Z 353.322,A -85,B 0,C 180,E1 -2944.271,E2 -2944.271} C_VEL
LIN {X 0,Y 560.701,Z 371.712,A -85,B 0,C 180,E1 -2946.548,E2 -2946.548} C_VEL
LIN {X 0,Y 560.278,Z 395.233,A -85,B 0,C 180,E1 -2949.437,E2 -2949.437} C_VEL
LIN {X 0,Y 560.248,Z 398.863,A -85,B 0,C 180,E1 -2949.881,E2 -2949.881} C_VEL
LIN {X 0,Y 561.84,Z 407.706,A -85,B 0,C 180,E1 -2950.065,E2 -2950.065} C_VEL
LIN {X 0,Y 561.234,Z 564.974,A -85,B 0,C 180,E1 -2952.145,E2 -2952.145} C_VEL
LIN {X 0,Y 561.075,Z 580.195,A -85,B 0,C 180,E1 -2952.491,E2 -2952.491} C_VEL
LIN {X 0,Y 560.834,Z 594.772,A -85,B 0,C 180,E1 -2952.966,E2 -2952.966} C_VEL
LIN {X 0,Y 560.63,Z 607.783,A -85,B 0,C 180,E1 -2953.522,E2 -2953.522} C_VEL
LIN {X 0,Y 560.319,Z 621.662,A -85,B 0,C 180,E1 -2954.261,E2 -2954.261} C_VEL
LIN {X 0,Y 560.023,Z 635.508,A -85,B 0,C 180,E1 -2955.173,E2 -2955.173} C_VEL
LIN {X 0,Y 559.723,Z 648.281,A -85,B 0,C 180,E1 -2956.197,E2 -2956.197} C_VEL
LIN {X 0,Y 559.517,Z 659.74,A -85,B 0,C 180,E1 -2957.301,E2 -2957.301} C_VEL
LIN {X 0,Y 559.306,Z 669.382,A -85,B 0,C 180,E1 -2958.401,E2 -2958.401} C_VEL
LIN {X 0,Y 559.169,Z 678.849,A -85,B 0,C 180,E1 -2959.682,E2 -2959.682} C_VEL
LIN {X 0,Y 559.003,Z 686.729,A -85,B 0,C 180,E1 -2960.957,E2 -2960.957} C_VEL
LIN {X 0,Y 558.921,Z 694.085,A -85,B 0,C 180,E1 -2962.412,E2 -2962.412} C_VEL
LIN {X 0,Y 558.859,Z 699.919,A -85,B 0,C 180,E1 -2963.863,E2 -2963.863} C_VEL
LIN {X 0,Y 558.787,Z 703.383,A -85,B 0,C 180,E1 -2964.948,E2 -2964.948} C_VEL
LIN {X 0,Y 558.819,Z 706.887,A -85,B 0,C 180,E1 -2966.394,E2 -2966.394} C_VEL
LIN {X 0,Y 558.744,Z 709.19,A -85,B 0,C 180,E1 -2967.836,E2 -2967.836} C_VEL
LIN {X 0,Y 558.737,Z 710.348,A -85,B 0,C 180,E1 -2969.278,E2 -2969.278} C_VEL
LIN {X 0,Y 558.737,Z 710.348,A -85,B 0,C 180,E1 -2970.72,E2 -2970.72} C_VEL
LIN {X 0,Y 558.744,Z 709.19,A -85,B 0,C 180,E1 -2972.161,E2 -2972.161} C_VEL
LIN {X 0,Y 558.819,Z 706.888,A -85,B 0,C 180,E1 -2973.604,E2 -2973.604} C_VEL
LIN {X 0,Y 558.787,Z 703.389,A -85,B 0,C 180,E1 -2975.05,E2 -2975.05} C_VEL
LIN {X 0,Y 558.869,Z 698.613,A -85,B 0,C 180,E1 -2976.497,E2 -2976.497} C_VEL
LIN {X 0,Y 558.949,Z 692.428,A -85,B 0,C 180,E1 -2977.949,E2 -2977.949} C_VEL
LIN {X 0,Y 559.004,Z 684.654,A -85,B 0,C 180,E1 -2979.405,E2 -2979.405} C_VEL
LIN {X 0,Y 559.216,Z 676.377,A -85,B 0,C 180,E1 -2980.682,E2 -2980.682} C_VEL
LIN {X 0,Y 559.36,Z 666.402,A -85,B 0,C 180,E1 -2981.964,E2 -2981.964} C_VEL
LIN {X 0,Y 559.595,Z 656.199,A -85,B 0,C 180,E1 -2983.064,E2 -2983.064} C_VEL
LIN {X 0,Y 559.859,Z 644.034,A -85,B 0,C 180,E1 -2984.168,E2 -2984.168} C_VEL
LIN {X 0,Y 560.121,Z 631.706,A -85,B 0,C 180,E1 -2985.099,E2 -2985.099} C_VEL
LIN {X 0,Y 560.357,Z 618.532,A -85,B 0,C 180,E1 -2985.922,E2 -2985.922} C_VEL
LIN {X 0,Y 560.663,Z 603.855,A -85,B 0,C 180,E1 -2986.662,E2 -2986.662} C_VEL
LIN {X 0,Y 560.943,Z 589.651,A -85,B 0,C 180,E1 -2987.216,E2 -2987.216} C_VEL
LIN {X 0,Y 561.139,Z 575.2,A -85,B 0,C 180,E1 -2987.636,E2 -2987.636} C_VEL
LIN {X 0,Y 561.23,Z 560.727,A -85,B 0,C 180,E1 -2987.922,E2 -2987.922} C_VEL
LIN {X 0,Y 561.79,Z 406.684,A -85,B 0,C 180,E1 -2989.951,E2 -2989.951} C_VEL
LIN {X 0,Y 560.235,Z 398.919,A -85,B 0,C 180,E1 -2990.112,E2 -2990.112} C_VEL
LIN {X 0,Y 560.643,Z 374.927,A -85,B 0,C 180,E1 -2993.061,E2 -2993.061} C_VEL
LIN {X 0,Y 561.028,Z 354.597,A -85,B 0,C 180,E1 -2995.585,E2 -2995.585} C_VEL
LIN {X 0,Y 559.73,Z 348.106,A -85,B 0,C 180,E1 -2996.469,E2 -2996.469} C_VEL
LIN {X 0,Y 559.123,Z 345.464,A -85,B 0,C 180,E1 -2996.863,E2 -2996.863} C_VEL
LIN {X 0,Y 559.133,Z 345.463,A -85,B 0,C 180,E1 -2999.855,E2 -2999.855} C_VEL
LIN {X 0,Y 559.143,Z 345.459,A -85,B 0,C 180,E1 -3002.714,E2 -3002.714} C_VEL
LIN {X 0,Y 559.106,Z 345.46,A -85,B 0,C 180,E1 -3005.324,E2 -3005.324} C_VEL
LIN {X 0,Y 559.115,Z 345.466,A -85,B 0,C 180,E1 -3008.017,E2 -3008.017} C_VEL
LIN {X 0,Y 559.116,Z 345.46,A -85,B 0,C 180,E1 -3010.814,E2 -3010.814} C_VEL
LIN {X 0,Y 559.115,Z 345.458,A -85,B 0,C 180,E1 -3013.193,E2 -3013.193} C_VEL
LIN {X 0,Y 559.111,Z 345.462,A -85,B 0,C 180,E1 -3015.763,E2 -3015.763} C_VEL
LIN {X 0,Y 559.108,Z 345.469,A -85,B 0,C 180,E1 -3018.225,E2 -3018.225} C_VEL
LIN {X 0,Y 559.156,Z 345.453,A -85,B 0,C 180,E1 -3021.192,E2 -3021.192} C_VEL
LIN {X 0,Y 559.101,Z 345.464,A -85,B 0,C 180,E1 -3023.786,E2 -3023.786} C_VEL
LIN {X 0,Y 559.145,Z 345.46,A -85,B 0,C 180,E1 -3026.424,E2 -3026.424} C_VEL
LIN {X 0,Y 559.136,Z 345.456,A -85,B 0,C 180,E1 -3028.98,E2 -3028.98} C_VEL
LIN {X 0,Y 559.093,Z 345.464,A -85,B 0,C 180,E1 -3031.63,E2 -3031.63} C_VEL
LIN {X 0,Y 559.111,Z 345.46,A -85,B 0,C 180,E1 -3034.699,E2 -3034.699} C_VEL
LIN {X 0,Y 559.095,Z 345.461,A -85,B 0,C 180,E1 -3037.066,E2 -3037.066} C_VEL
LIN {X 0,Y 559.146,Z 345.455,A -85,B 0,C 180,E1 -3039.394,E2 -3039.394} C_VEL
LIN {X 0,Y 559.105,Z 345.463,A -85,B 0,C 180,E1 -3041.684,E2 -3041.684} C_VEL
LIN {X 0,Y 559.115,Z 345.46,A -85,B 0,C 180,E1 -3044.695,E2 -3044.695} C_VEL
LIN {X 0,Y 559.125,Z 345.457,A -85,B 0,C 180,E1 -3046.924,E2 -3046.924} C_VEL
LIN {X 0,Y 559.173,Z 345.451,A -85,B 0,C 180,E1 -3049.133,E2 -3049.133} C_VEL
LIN {X 0,Y 559.152,Z 345.464,A -85,B 0,C 180,E1 -3052.053,E2 -3052.053} C_VEL
LIN {X 0,Y 559.214,Z 345.446,A -85,B 0,C 180,E1 -3054.953,E2 -3054.953} C_VEL
LIN {X 0,Y 559.236,Z 345.45,A -85,B 0,C 180,E1 -3057.84,E2 -3057.84} C_VEL
LIN {X 0,Y 559.239,Z 345.453,A -85,B 0,C 180,E1 -3060,E2 -3060} C_VEL
LIN {X 0,Y 559.191,Z 345.449,A -85,B 0,C 180,E1 -3062.882,E2 -3062.882} C_VEL
LIN {X 0,Y 559.192,Z 345.455,A -85,B 0,C 180,E1 -3065.771,E2 -3065.771} C_VEL
LIN {X 0,Y 559.143,Z 345.456,A -85,B 0,C 180,E1 -3068.675,E2 -3068.675} C_VEL
LIN {X 0,Y 559.14,Z 345.46,A -85,B 0,C 180,E1 -3071.602,E2 -3071.602} C_VEL
LIN {X 0,Y 559.166,Z 345.453,A -85,B 0,C 180,E1 -3074.588,E2 -3074.588} C_VEL
LIN {X 0,Y 559.1,Z 345.464,A -85,B 0,C 180,E1 -3077.559,E2 -3077.559} C_VEL
LIN {X 0,Y 559.145,Z 345.463,A -85,B 0,C 180,E1 -3079.839,E2 -3079.839} C_VEL
LIN {X 0,Y 559.114,Z 345.465,A -85,B 0,C 180,E1 -3082.154,E2 -3082.154} C_VEL
LIN {X 0,Y 559.124,Z 345.458,A -85,B 0,C 180,E1 -3085.179,E2 -3085.179} C_VEL
LIN {X 0,Y 559.091,Z 345.468,A -85,B 0,C 180,E1 -3087.717,E2 -3087.717} C_VEL
LIN {X 0,Y 559.112,Z 345.46,A -85,B 0,C 180,E1 -3090.584,E2 -3090.584} C_VEL
LIN {X 0,Y 558.456,Z 345.542,A -85,B 0,C 180,E1 -3091.186,E2 -3091.186} C_VEL
LIN {X 0,Y 555.6,Z 345.902,A -85,B 0,C 180,E1 -3092.162,E2 -3092.162} C_VEL
LIN {X 0,Y 553.189,Z 346.199,A -85,B 0,C 180,E1 -3092.948,E2 -3092.948} C_VEL
LIN {X 0,Y 552.167,Z 346.329,A -85,B 0,C 180,E1 -3093.554,E2 -3093.554} C_VEL
LIN {X 0,Y 552.092,Z 346.336,A -85,B 0,C 180,E1 -3093.76,E2 -3093.76} C_VEL
LIN {X 0,Y 552.057,Z 346.338,A -85,B 0,C 180,E1 -3096.751,E2 -3096.751} C_VEL
LIN {X 0,Y 552.115,Z 346.335,A -85,B 0,C 180,E1 -3099.529,E2 -3099.529} C_VEL
LIN {X 0,Y 552.076,Z 346.337,A -85,B 0,C 180,E1 -3102.431,E2 -3102.431} C_VEL
LIN {X 0,Y 552.065,Z 346.342,A -85,B 0,C 180,E1 -3105.561,E2 -3105.561} C_VEL
LIN {X 0,Y 552.1,Z 346.338,A -85,B 0,C 180,E1 -3107.589,E2 -3107.589} C_VEL
LIN {X 0,Y 552.118,Z 346.331,A -85,B 0,C 180,E1 -3110.474,E2 -3110.474} C_VEL
LIN {X 0,Y 552.089,Z 346.336,A -85,B 0,C 180,E1 -3113.32,E2 -3113.32} C_VEL
LIN {X 0,Y 552.109,Z 346.339,A -85,B 0,C 180,E1 -3115.94,E2 -3115.94} C_VEL
LIN {X 0,Y 552.116,Z 346.331,A -85,B 0,C 180,E1 -3118.542,E2 -3118.542} C_VEL
LIN {X 0,Y 552.072,Z 346.34,A -85,B 0,C 180,E1 -3121.449,E2 -3121.449} C_VEL
LIN {X 0,Y 552.077,Z 346.337,A -85,B 0,C 180,E1 -3124.355,E2 -3124.355} C_VEL
LIN {X 0,Y 552.09,Z 346.333,A -85,B 0,C 180,E1 -3126.759,E2 -3126.759} C_VEL
LIN {X 0,Y 552.114,Z 346.332,A -85,B 0,C 180,E1 -3129.121,E2 -3129.121} C_VEL
LIN {X 0,Y 552.082,Z 346.34,A -85,B 0,C 180,E1 -3131.444,E2 -3131.444} C_VEL
LIN {X 0,Y 552.084,Z 346.344,A -85,B 0,C 180,E1 -3133.738,E2 -3133.738} C_VEL
LIN {X 0,Y 552.125,Z 346.334,A -85,B 0,C 180,E1 -3136.005,E2 -3136.005} C_VEL
LIN {X 0,Y 552.161,Z 346.325,A -85,B 0,C 180,E1 -3138.995,E2 -3138.995} C_VEL
LIN {X 0,Y 552.113,Z 346.336,A -85,B 0,C 180,E1 -3141.952,E2 -3141.952} C_VEL
LIN {X 0,Y 552.212,Z 346.319,A -85,B 0,C 180,E1 -3144.89,E2 -3144.89} C_VEL
LIN {X 0,Y 552.223,Z 346.324,A -85,B 0,C 180,E1 -3147.813,E2 -3147.813} C_VEL
LIN {X 0,Y 552.226,Z 346.321,A -85,B 0,C 180,E1 -3150.001,E2 -3150.001} C_VEL
LIN {X 0,Y 552.184,Z 346.322,A -85,B 0,C 180,E1 -3152.919,E2 -3152.919} C_VEL
LIN {X 0,Y 552.187,Z 346.328,A -85,B 0,C 180,E1 -3155.845,E2 -3155.845} C_VEL
LIN {X 0,Y 552.137,Z 346.328,A -85,B 0,C 180,E1 -3158.787,E2 -3158.787} C_VEL
LIN {X 0,Y 552.158,Z 346.333,A -85,B 0,C 180,E1 -3161.752,E2 -3161.752} C_VEL
LIN {X 0,Y 552.134,Z 346.328,A -85,B 0,C 180,E1 -3164.749,E2 -3164.749} C_VEL
LIN {X 0,Y 552.082,Z 346.341,A -85,B 0,C 180,E1 -3167.79,E2 -3167.79} C_VEL
LIN {X 0,Y 552.129,Z 346.331,A -85,B 0,C 180,E1 -3170.102,E2 -3170.102} C_VEL
LIN {X 0,Y 552.089,Z 346.334,A -85,B 0,C 180,E1 -3172.452,E2 -3172.452} C_VEL
LIN {X 0,Y 552.09,Z 346.34,A -85,B 0,C 180,E1 -3175.335,E2 -3175.335} C_VEL
LIN {X 0,Y 552.069,Z 346.338,A -85,B 0,C 180,E1 -3178.101,E2 -3178.101} C_VEL
LIN {X 0,Y 552.098,Z 346.332,A -85,B 0,C 180,E1 -3180.61,E2 -3180.61} C_VEL
LIN {X 0,Y 552.119,Z 346.334,A -85,B 0,C 180,E1 -3183.186,E2 -3183.186} C_VEL
LIN {X 0,Y 552.077,Z 346.341,A -85,B 0,C 180,E1 -3185.845,E2 -3185.845} C_VEL
LIN {X 0,Y 552.119,Z 346.331,A -85,B 0,C 180,E1 -3188.59,E2 -3188.59} C_VEL
LIN {X 0,Y 552.116,Z 346.34,A -85,B 0,C 180,E1 -3191.447,E2 -3191.447} C_VEL
LIN {X 0,Y 552.087,Z 346.337,A -85,B 0,C 180,E1 -3194.53,E2 -3194.53} C_VEL
LIN {X 0,Y 552.136,Z 346.514,A -85,B 0,C 180,E1 -3197.181,E2 -3197.181} C_VEL
LIN {X 0,Y 553.352,Z 352.723,A -85,B 0,C 180,E1 -3198.157,E2 -3198.157} C_VEL
LIN {X 0,Y 553.112,Z 369.626,A -85,B 0,C 180,E1 -3200.625,E2 -3200.625} C_VEL
LIN {X 0,Y 553.086,Z 369.981,A -85,B 0,C 180,E1 -3200.675,E2 -3200.675} C_VEL
LIN {X 0,Y 555.117,Z 380.22,A -85,B 0,C 180,E1 -3200.892,E2 -3200.892} C_VEL
LIN {X 0,Y 554.469,Z 534.941,A -85,B 0,C 180,E1 -3202.966,E2 -3202.966} C_VEL
LIN {X 0,Y 554.241,Z 551.404,A -85,B 0,C 180,E1 -3203.347,E2 -3203.347} C_VEL
LIN {X 0,Y 554.002,Z 566.172,A -85,B 0,C 180,E1 -3203.85,E2 -3203.85} C_VEL
LIN {X 0,Y 553.717,Z 578.767,A -85,B 0,C 180,E1 -3204.409,E2 -3204.409} C_VEL
LIN {X 0,Y 553.438,Z 590.432,A -85,B 0,C 180,E1 -3205.038,E2 -3205.038} C_VEL
LIN {X 0,Y 553.173,Z 601.881,A -85,B 0,C 180,E1 -3205.763,E2 -3205.763} C_VEL
LIN {X 0,Y 552.882,Z 614.744,A -85,B 0,C 180,E1 -3206.757,E2 -3206.757} C_VEL
LIN {X 0,Y 552.588,Z 626.309,A -85,B 0,C 180,E1 -3207.828,E2 -3207.828} C_VEL
LIN {X 0,Y 552.337,Z 636.84,A -85,B 0,C 180,E1 -3208.98,E2 -3208.98} C_VEL
LIN {X 0,Y 552.158,Z 646.412,A -85,B 0,C 180,E1 -3210.238,E2 -3210.238} C_VEL
LIN {X 0,Y 551.992,Z 654.342,A -85,B 0,C 180,E1 -3211.465,E2 -3211.465} C_VEL
LIN {X 0,Y 551.865,Z 661.042,A -85,B 0,C 180,E1 -3212.712,E2 -3212.712} C_VEL
LIN {X 0,Y 551.8,Z 666.54,A -85,B 0,C 180,E1 -3213.934,E2 -3213.934} C_VEL
LIN {X 0,Y 551.74,Z 672.249,A -85,B 0,C 180,E1 -3215.545,E2 -3215.545} C_VEL
LIN {X 0,Y 551.701,Z 675.466,A -85,B 0,C 180,E1 -3216.74,E2 -3216.74} C_VEL
LIN {X 0,Y 551.678,Z 678.639,A -85,B 0,C 180,E1 -3218.431,E2 -3218.431} C_VEL
LIN {X 0,Y 551.637,Z 680.119,A -85,B 0,C 180,E1 -3219.88,E2 -3219.88} C_VEL
LIN {X 0,Y 551.645,Z 680.42,A -85,B 0,C 180,E1 -3221.427,E2 -3221.427} C_VEL
LIN {X 0,Y 551.668,Z 679.51,A -85,B 0,C 180,E1 -3222.962,E2 -3222.962} C_VEL
LIN {X 0,Y 551.627,Z 677.296,A -85,B 0,C 180,E1 -3224.481,E2 -3224.481} C_VEL
LIN {X 0,Y 551.711,Z 673.879,A -85,B 0,C 180,E1 -3225.993,E2 -3225.993} C_VEL
LIN {X 0,Y 551.778,Z 669.079,A -85,B 0,C 180,E1 -3227.495,E2 -3227.495} C_VEL
LIN {X 0,Y 551.853,Z 662.934,A -85,B 0,C 180,E1 -3228.987,E2 -3228.987} C_VEL
LIN {X 0,Y 551.96,Z 656.255,A -85,B 0,C 180,E1 -3230.287,E2 -3230.287} C_VEL
LIN {X 0,Y 552.097,Z 648.306,A -85,B 0,C 180,E1 -3231.582,E2 -3231.582} C_VEL
LIN {X 0,Y 552.328,Z 639.127,A -85,B 0,C 180,E1 -3232.826,E2 -3232.826} C_VEL
LIN {X 0,Y 552.56,Z 629.074,A -85,B 0,C 180,E1 -3233.977,E2 -3233.977} C_VEL
LIN {X 0,Y 552.757,Z 617.741,A -85,B 0,C 180,E1 -3235.076,E2 -3235.076} C_VEL
LIN {X 0,Y 553.156,Z 603.953,A -85,B 0,C 180,E1 -3236.175,E2 -3236.175} C_VEL
LIN {X 0,Y 553.453,Z 591.502,A -85,B 0,C 180,E1 -3236.997,E2 -3236.997} C_VEL
LIN {X 0,Y 553.76,Z 577.924,A -85,B 0,C 180,E1 -3237.727,E2 -3237.727} C_VEL
LIN {X 0,Y 554.081,Z 562.907,A -85,B 0,C 180,E1 -3238.364,E2 -3238.364} C_VEL
LIN {X 0,Y 554.312,Z 546.854,A -85,B 0,C 180,E1 -3238.865,E2 -3238.865} C_VEL
LIN {X 0,Y 554.523,Z 531.367,A -85,B 0,C 180,E1 -3239.183,E2 -3239.183} C_VEL
LIN {X 0,Y 555.126,Z 379.728,A -85,B 0,C 180,E1 -3241.204,E2 -3241.204} C_VEL
LIN {X 0,Y 553.108,Z 369.903,A -85,B 0,C 180,E1 -3241.429,E2 -3241.429} C_VEL
LIN {X 0,Y 553.467,Z 353.564,A -85,B 0,C 180,E1 -3243.822,E2 -3243.822} C_VEL
LIN {X 0,Y 552.204,Z 346.328,A -85,B 0,C 180,E1 -3244.974,E2 -3244.974} C_VEL
LIN {X 0,Y 552.174,Z 346.328,A -85,B 0,C 180,E1 -3247.312,E2 -3247.312} C_VEL
LIN {X 0,Y 552.101,Z 346.341,A -85,B 0,C 180,E1 -3250.266,E2 -3250.266} C_VEL
LIN {X 0,Y 552.141,Z 346.336,A -85,B 0,C 180,E1 -3252.497,E2 -3252.497} C_VEL
LIN {X 0,Y 552.14,Z 346.335,A -85,B 0,C 180,E1 -3254.748,E2 -3254.748} C_VEL
LIN {X 0,Y 552.095,Z 346.336,A -85,B 0,C 180,E1 -3257.789,E2 -3257.789} C_VEL
LIN {X 0,Y 552.128,Z 346.336,A -85,B 0,C 180,E1 -3260.101,E2 -3260.101} C_VEL
LIN {X 0,Y 552.093,Z 346.342,A -85,B 0,C 180,E1 -3262.451,E2 -3262.451} C_VEL
LIN {X 0,Y 552.084,Z 346.335,A -85,B 0,C 180,E1 -3265.333,E2 -3265.333} C_VEL
LIN {X 0,Y 552.056,Z 346.346,A -85,B 0,C 180,E1 -3268.101,E2 -3268.101} C_VEL
LIN {X 0,Y 552.092,Z 346.338,A -85,B 0,C 180,E1 -3270.61,E2 -3270.61} C_VEL
LIN {X 0,Y 552.098,Z 346.334,A -85,B 0,C 180,E1 -3273.187,E2 -3273.187} C_VEL
LIN {X 0,Y 552.066,Z 346.343,A -85,B 0,C 180,E1 -3275.845,E2 -3275.845} C_VEL
LIN {X 0,Y 552.114,Z 346.331,A -85,B 0,C 180,E1 -3279.059,E2 -3279.059} C_VEL
LIN {X 0,Y 552.081,Z 346.34,A -85,B 0,C 180,E1 -3282.409,E2 -3282.409} C_VEL
LIN {X 0,Y 552.064,Z 346.34,A -85,B 0,C 180,E1 -3285.558,E2 -3285.558} C_VEL
LIN {X 0,Y 552.051,Z 346.341,A -85,B 0,C 180,E1 -3288.547,E2 -3288.547} C_VEL
LIN {X 0,Y 552.088,Z 346.338,A -85,B 0,C 180,E1 -3291.408,E2 -3291.408} C_VEL
LIN {X 0,Y 552.06,Z 346.341,A -85,B 0,C 180,E1 -3294.563,E2 -3294.563} C_VEL
LIN {X 0,Y 552.098,Z 346.338,A -85,B 0,C 180,E1 -3297.156,E2 -3297.156} C_VEL
LIN {X 0,Y 552.088,Z 346.345,A -85,B 0,C 180,E1 -3299.955,E2 -3299.955} C_VEL
LIN {X 0,Y 552.06,Z 346.347,A -85,B 0,C 180,E1 -3302.973,E2 -3302.973} C_VEL
LIN {X 0,Y 554.103,Z 355.391,A -85,B 0,C 180,E1 -3304.228,E2 -3304.228} C_VEL
LIN {X 0,Y 553.795,Z 374.625,A -85,B 0,C 180,E1 -3306.634,E2 -3306.634} C_VEL
LIN {X 0,Y 553.364,Z 398.741,A -85,B 0,C 180,E1 -3309.605,E2 -3309.605} C_VEL
LIN {X 0,Y 555.181,Z 408.505,A -85,B 0,C 180,E1 -3309.826,E2 -3309.826} C_VEL
LIN {X 0,Y 554.471,Z 565.076,A -85,B 0,C 180,E1 -3311.922,E2 -3311.922} C_VEL
LIN {X 0,Y 554.296,Z 580.671,A -85,B 0,C 180,E1 -3312.283,E2 -3312.283} C_VEL
LIN {X 0,Y 554.009,Z 596.013,A -85,B 0,C 180,E1 -3312.797,E2 -3312.797} C_VEL
LIN {X 0,Y 553.761,Z 609.759,A -85,B 0,C 180,E1 -3313.407,E2 -3313.407} C_VEL
LIN {X 0,Y 553.407,Z 623.236,A -85,B 0,C 180,E1 -3314.154,E2 -3314.154} C_VEL
LIN {X 0,Y 553.086,Z 636.289,A -85,B 0,C 180,E1 -3315.04,E2 -3315.04} C_VEL
LIN {X 0,Y 552.781,Z 648.282,A -85,B 0,C 180,E1 -3316.02,E2 -3316.02} C_VEL
LIN {X 0,Y 552.53,Z 659.74,A -85,B 0,C 180,E1 -3317.138,E2 -3317.138} C_VEL
LIN {X 0,Y 552.254,Z 670.43,A -85,B 0,C 180,E1 -3318.382,E2 -3318.382} C_VEL
LIN {X 0,Y 552.125,Z 678.849,A -85,B 0,C 180,E1 -3319.548,E2 -3319.548} C_VEL
LIN {X 0,Y 551.958,Z 686.73,A -85,B 0,C 180,E1 -3320.841,E2 -3320.841} C_VEL
LIN {X 0,Y 551.838,Z 694.086,A -85,B 0,C 180,E1 -3322.314,E2 -3322.314} C_VEL
LIN {X 0,Y 551.759,Z 699.603,A -85,B 0,C 180,E1 -3323.69,E2 -3323.69} C_VEL
LIN {X 0,Y 551.713,Z 703.383,A -85,B 0,C 180,E1 -3324.883,E2 -3324.883} C_VEL
LIN {X 0,Y 551.731,Z 706.887,A -85,B 0,C 180,E1 -3326.347,E2 -3326.347} C_VEL
LIN {X 0,Y 551.654,Z 709.19,A -85,B 0,C 180,E1 -3327.809,E2 -3327.809} C_VEL
LIN {X 0,Y 551.637,Z 710.348,A -85,B 0,C 180,E1 -3329.269,E2 -3329.269} C_VEL
LIN {X 0,Y 551.637,Z 710.348,A -85,B 0,C 180,E1 -3330.729,E2 -3330.729} C_VEL
LIN {X 0,Y 551.654,Z 709.189,A -85,B 0,C 180,E1 -3332.189,E2 -3332.189} C_VEL
LIN {X 0,Y 551.73,Z 706.888,A -85,B 0,C 180,E1 -3333.651,E2 -3333.651} C_VEL
LIN {X 0,Y 551.713,Z 703.39,A -85,B 0,C 180,E1 -3335.115,E2 -3335.115} C_VEL
LIN {X 0,Y 551.819,Z 698.613,A -85,B 0,C 180,E1 -3336.581,E2 -3336.581} C_VEL
LIN {X 0,Y 551.875,Z 692.427,A -85,B 0,C 180,E1 -3338.051,E2 -3338.051} C_VEL
LIN {X 0,Y 551.95,Z 684.653,A -85,B 0,C 180,E1 -3339.527,E2 -3339.527} C_VEL
LIN {X 0,Y 552.182,Z 676.376,A -85,B 0,C 180,E1 -3340.819,E2 -3340.819} C_VEL
LIN {X 0,Y 552.35,Z 666.402,A -85,B 0,C 180,E1 -3342.118,E2 -3342.118} C_VEL
LIN {X 0,Y 552.607,Z 656.198,A -85,B 0,C 180,E1 -3343.232,E2 -3343.232} C_VEL
LIN {X 0,Y 552.905,Z 644.034,A -85,B 0,C 180,E1 -3344.35,E2 -3344.35} C_VEL
LIN {X 0,Y 553.245,Z 631.46,A -85,B 0,C 180,E1 -3345.309,E2 -3345.309} C_VEL
LIN {X 0,Y 553.507,Z 618.53,A -85,B 0,C 180,E1 -3346.125,E2 -3346.125} C_VEL
LIN {X 0,Y 553.865,Z 603.852,A -85,B 0,C 180,E1 -3346.872,E2 -3346.872} C_VEL
LIN {X 0,Y 554.15,Z 589.65,A -85,B 0,C 180,E1 -3347.434,E2 -3347.434} C_VEL
LIN {X 0,Y 554.351,Z 574.561,A -85,B 0,C 180,E1 -3347.876,E2 -3347.876} C_VEL
LIN {X 0,Y 554.516,Z 559.219,A -85,B 0,C 180,E1 -3348.17,E2 -3348.17} C_VEL
LIN {X 0,Y 555.058,Z 407.591,A -85,B 0,C 180,E1 -3350.191,E2 -3350.191} C_VEL
LIN {X 0,Y 553.345,Z 398.833,A -85,B 0,C 180,E1 -3350.384,E2 -3350.384} C_VEL
LIN {X 0,Y 553.802,Z 374.781,A -85,B 0,C 180,E1 -3353.363,E2 -3353.363} C_VEL
LIN {X 0,Y 554.19,Z 355.492,A -85,B 0,C 180,E1 -3355.791,E2 -3355.791} C_VEL
LIN {X 0,Y 552.06,Z 346.344,A -85,B 0,C 180,E1 -3357.093,E2 -3357.093} C_VEL
LIN {X 0,Y 552.103,Z 346.34,A -85,B 0,C 180,E1 -3360.048,E2 -3360.048} C_VEL
LIN {X 0,Y 552.102,Z 346.335,A -85,B 0,C 180,E1 -3362.844,E2 -3362.844} C_VEL
LIN {X 0,Y 552.054,Z 346.34,A -85,B 0,C 180,E1 -3365.436,E2 -3365.436} C_VEL
LIN {X 0,Y 552.078,Z 346.341,A -85,B 0,C 180,E1 -3367.883,E2 -3367.883} C_VEL
LIN {X 0,Y 552.081,Z 346.34,A -85,B 0,C 180,E1 -3370.482,E2 -3370.482} C_VEL
LIN {X 0,Y 552.081,Z 346.335,A -85,B 0,C 180,E1 -3373.48,E2 -3373.48} C_VEL
LIN {X 0,Y 552.06,Z 346.341,A -85,B 0,C 180,E1 -3376.572,E2 -3376.572} C_VEL
LIN {X 0,Y 552.091,Z 346.337,A -85,B 0,C 180,E1 -3379.797,E2 -3379.797} C_VEL
LIN {X 0,Y 552.069,Z 346.343,A -85,B 0,C 180,E1 -3382.334,E2 -3382.334} C_VEL
LIN {X 0,Y 552.061,Z 346.337,A -85,B 0,C 180,E1 -3385.049,E2 -3385.049} C_VEL
LIN {X 0,Y 552.098,Z 346.336,A -85,B 0,C 180,E1 -3387.68,E2 -3387.68} C_VEL
LIN {X 0,Y 552.067,Z 346.345,A -85,B 0,C 180,E1 -3390.233,E2 -3390.233} C_VEL
LIN {X 0,Y 552.062,Z 346.337,A -85,B 0,C 180,E1 -3393.012,E2 -3393.012} C_VEL
LIN {X 0,Y 552.067,Z 346.344,A -85,B 0,C 180,E1 -3395.96,E2 -3395.96} C_VEL
LIN {X 0,Y 552.089,Z 346.334,A -85,B 0,C 180,E1 -3399.119,E2 -3399.119} C_VEL
LIN {X 0,Y 552.066,Z 346.338,A -85,B 0,C 180,E1 -3401.443,E2 -3401.443} C_VEL
LIN {X 0,Y 552.073,Z 346.339,A -85,B 0,C 180,E1 -3404.494,E2 -3404.494} C_VEL
LIN {X 0,Y 552.088,Z 346.335,A -85,B 0,C 180,E1 -3406.754,E2 -3406.754} C_VEL
LIN {X 0,Y 552.142,Z 346.327,A -85,B 0,C 180,E1 -3408.993,E2 -3408.993} C_VEL
LIN {X 0,Y 552.113,Z 346.339,A -85,B 0,C 180,E1 -3411.951,E2 -3411.951} C_VEL
LIN {X 0,Y 552.191,Z 346.321,A -85,B 0,C 180,E1 -3414.889,E2 -3414.889} C_VEL
LIN {X 0,Y 552.206,Z 346.326,A -85,B 0,C 180,E1 -3417.812,E2 -3417.812} C_VEL
LIN {X 0,Y 552.208,Z 346.329,A -85,B 0,C 180,E1 -3420,E2 -3420} C_VEL
LIN {X 0,Y 552.158,Z 346.325,A -85,B 0,C 180,E1 -3422.919,E2 -3422.919} C_VEL
LIN {X 0,Y 552.163,Z 346.332,A -85,B 0,C 180,E1 -3425.844,E2 -3425.844} C_VEL
LIN {X 0,Y 552.114,Z 346.331,A -85,B 0,C 180,E1 -3428.787,E2 -3428.787} C_VEL
LIN {X 0,Y 552.086,Z 346.34,A -85,B 0,C 180,E1 -3431.752,E2 -3431.752} C_VEL
LIN {X 0,Y 552.113,Z 346.331,A -85,B 0,C 180,E1 -3434.749,E2 -3434.749} C_VEL
LIN {X 0,Y 552.064,Z 346.344,A -85,B 0,C 180,E1 -3437.79,E2 -3437.79} C_VEL
LIN {X 0,Y 552.104,Z 346.339,A -85,B 0,C 180,E1 -3440.102,E2 -3440.102} C_VEL
LIN {X 0,Y 552.067,Z 346.339,A -85,B 0,C 180,E1 -3442.452,E2 -3442.452} C_VEL
LIN {X 0,Y 552.066,Z 346.338,A -85,B 0,C 180,E1 -3445.334,E2 -3445.334} C_VEL
LIN {X 0,Y 552.04,Z 346.346,A -85,B 0,C 180,E1 -3448.103,E2 -3448.103} C_VEL
LIN {X 0,Y 552.077,Z 346.336,A -85,B 0,C 180,E1 -3450.611,E2 -3450.611} C_VEL
LIN {X 0,Y 552.1,Z 346.333,A -85,B 0,C 180,E1 -3453.187,E2 -3453.187} C_VEL
LIN {X 0,Y 552.092,Z 346.336,A -85,B 0,C 180,E1 -3453.76,E2 -3453.76} C_VEL
LIN {X 0,Y 551.442,Z 346.421,A -85,B 0,C 180,E1 -3454.368,E2 -3454.368} C_VEL
LIN {X 0,Y 548.575,Z 346.777,A -85,B 0,C 180,E1 -3455.356,E2 -3455.356} C_VEL
LIN {X 0,Y 546.138,Z 347.08,A -85,B 0,C 180,E1 -3456.151,E2 -3456.151} C_VEL
LIN {X 0,Y 545.089,Z 347.206,A -85,B 0,C 180,E1 -3456.765,E2 -3456.765} C_VEL
LIN {X 0,Y 545.003,Z 347.216,A -85,B 0,C 180,E1 -3456.973,E2 -3456.973} C_VEL
LIN {X 0,Y 545.061,Z 347.211,A -85,B 0,C 180,E1 -3459.321,E2 -3459.321} C_VEL
LIN {X 0,Y 545.026,Z 347.219,A -85,B 0,C 180,E1 -3462.108,E2 -3462.108} C_VEL
LIN {X 0,Y 545.012,Z 347.216,A -85,B 0,C 180,E1 -3465.173,E2 -3465.173} C_VEL
LIN {X 0,Y 545.043,Z 347.22,A -85,B 0,C 180,E1 -3467.896,E2 -3467.896} C_VEL
LIN {X 0,Y 545.068,Z 347.208,A -85,B 0,C 180,E1 -3470.819,E2 -3470.819} C_VEL
LIN {X 0,Y 545.024,Z 347.221,A -85,B 0,C 180,E1 -3473.62,E2 -3473.62} C_VEL
LIN {X 0,Y 545.051,Z 347.212,A -85,B 0,C 180,E1 -3476.329,E2 -3476.329} C_VEL
LIN {X 0,Y 545.058,Z 347.21,A -85,B 0,C 180,E1 -3478.953,E2 -3478.953} C_VEL
LIN {X 0,Y 545.033,Z 347.218,A -85,B 0,C 180,E1 -3481.505,E2 -3481.505} C_VEL
LIN {X 0,Y 545.031,Z 347.213,A -85,B 0,C 180,E1 -3484.506,E2 -3484.506} C_VEL
LIN {X 0,Y 545.031,Z 347.215,A -85,B 0,C 180,E1 -3487.243,E2 -3487.243} C_VEL
LIN {X 0,Y 545.115,Z 347.203,A -85,B 0,C 180,E1 -3490.416,E2 -3490.416} C_VEL
LIN {X 0,Y 545.035,Z 347.219,A -85,B 0,C 180,E1 -3493.521,E2 -3493.521} C_VEL
LIN {X 0,Y 545.081,Z 347.215,A -85,B 0,C 180,E1 -3495.821,E2 -3495.821} C_VEL
LIN {X 0,Y 545.117,Z 347.202,A -85,B 0,C 180,E1 -3498.851,E2 -3498.851} C_VEL
LIN {X 0,Y 545.071,Z 347.215,A -85,B 0,C 180,E1 -3501.847,E2 -3501.847} C_VEL
LIN {X 0,Y 545.17,Z 347.196,A -85,B 0,C 180,E1 -3504.824,E2 -3504.824} C_VEL
LIN {X 0,Y 545.194,Z 347.2,A -85,B 0,C 180,E1 -3507.785,E2 -3507.785} C_VEL
LIN {X 0,Y 545.194,Z 347.197,A -85,B 0,C 180,E1 -3510.001,E2 -3510.001} C_VEL
LIN {X 0,Y 545.152,Z 347.199,A -85,B 0,C 180,E1 -3512.957,E2 -3512.957} C_VEL
LIN {X 0,Y 545.137,Z 347.205,A -85,B 0,C 180,E1 -3515.921,E2 -3515.921} C_VEL
LIN {X 0,Y 545.098,Z 347.205,A -85,B 0,C 180,E1 -3518.901,E2 -3518.901} C_VEL
LIN {X 0,Y 545.1,Z 347.209,A -85,B 0,C 180,E1 -3521.906,E2 -3521.906} C_VEL
LIN {X 0,Y 545.085,Z 347.207,A -85,B 0,C 180,E1 -3524.945,E2 -3524.945} C_VEL
LIN {X 0,Y 545.053,Z 347.213,A -85,B 0,C 180,E1 -3528.028,E2 -3528.028} C_VEL
LIN {X 0,Y 545.096,Z 347.205,A -85,B 0,C 180,E1 -3530.373,E2 -3530.373} C_VEL
LIN {X 0,Y 545.078,Z 347.217,A -85,B 0,C 180,E1 -3533.56,E2 -3533.56} C_VEL
LIN {X 0,Y 545.061,Z 347.21,A -85,B 0,C 180,E1 -3536.827,E2 -3536.827} C_VEL
LIN {X 0,Y 545.035,Z 347.219,A -85,B 0,C 180,E1 -3539.341,E2 -3539.341} C_VEL
LIN {X 0,Y 545.06,Z 347.213,A -85,B 0,C 180,E1 -3541.915,E2 -3541.915} C_VEL
LIN {X 0,Y 545.056,Z 347.21,A -85,B 0,C 180,E1 -3544.566,E2 -3544.566} C_VEL
LIN {X 0,Y 545.036,Z 347.221,A -85,B 0,C 180,E1 -3547.305,E2 -3547.305} C_VEL
LIN {X 0,Y 545.07,Z 347.211,A -85,B 0,C 180,E1 -3550.143,E2 -3550.143} C_VEL
LIN {X 0,Y 545.051,Z 347.217,A -85,B 0,C 180,E1 -3553.11,E2 -3553.11} C_VEL
LIN {X 0,Y 545.051,Z 347.218,A -85,B 0,C 180,E1 -3556.227,E2 -3556.227} C_VEL
LIN {X 0,Y 545.065,Z 347.266,A -85,B 0,C 180,E1 -3556.946,E2 -3556.946} C_VEL
LIN {X 0,Y 546.471,Z 354.048,A -85,B 0,C 180,E1 -3558.028,E2 -3558.028} C_VEL
LIN {X 0,Y 546.251,Z 368.73,A -85,B 0,C 180,E1 -3560.202,E2 -3560.202} C_VEL
LIN {X 0,Y 546.232,Z 370.233,A -85,B 0,C 180,E1 -3560.41,E2 -3560.41} C_VEL
LIN {X 0,Y 548.462,Z 381.063,A -85,B 0,C 180,E1 -3560.651,E2 -3560.651} C_VEL
LIN {X 0,Y 547.78,Z 534.336,A -85,B 0,C 180,E1 -3562.726,E2 -3562.726} C_VEL
LIN {X 0,Y 547.517,Z 550.412,A -85,B 0,C 180,E1 -3563.095,E2 -3563.095} C_VEL
LIN {X 0,Y 547.226,Z 564.398,A -85,B 0,C 180,E1 -3563.559,E2 -3563.559} C_VEL
LIN {X 0,Y 546.922,Z 577.647,A -85,B 0,C 180,E1 -3564.14,E2 -3564.14} C_VEL
LIN {X 0,Y 546.636,Z 589.227,A -85,B 0,C 180,E1 -3564.76,E2 -3564.76} C_VEL
LIN {X 0,Y 546.287,Z 601.273,A -85,B 0,C 180,E1 -3565.524,E2 -3565.524} C_VEL
LIN {X 0,Y 545.976,Z 614.129,A -85,B 0,C 180,E1 -3566.52,E2 -3566.52} C_VEL
LIN {X 0,Y 545.615,Z 626.587,A -85,B 0,C 180,E1 -3567.686,E2 -3567.686} C_VEL
LIN {X 0,Y 545.376,Z 636.251,A -85,B 0,C 180,E1 -3568.756,E2 -3568.756} C_VEL
LIN {X 0,Y 545.147,Z 645.938,A -85,B 0,C 180,E1 -3570.029,E2 -3570.029} C_VEL
LIN {X 0,Y 544.951,Z 653.985,A -85,B 0,C 180,E1 -3571.28,E2 -3571.28} C_VEL
LIN {X 0,Y 544.804,Z 661.236,A -85,B 0,C 180,E1 -3572.645,E2 -3572.645} C_VEL
LIN {X 0,Y 544.708,Z 667.114,A -85,B 0,C 180,E1 -3573.98,E2 -3573.98} C_VEL
LIN {X 0,Y 544.648,Z 672.656,A -85,B 0,C 180,E1 -3575.611,E2 -3575.611} C_VEL
LIN {X 0,Y 544.567,Z 676.65,A -85,B 0,C 180,E1 -3577.221,E2 -3577.221} C_VEL
LIN {X 0,Y 544.562,Z 679.187,A -85,B 0,C 180,E1 -3578.816,E2 -3578.816} C_VEL
LIN {X 0,Y 544.588,Z 680.351,A -85,B 0,C 180,E1 -3580.405,E2 -3580.405} C_VEL
LIN {X 0,Y 544.553,Z 680.28,A -85,B 0,C 180,E1 -3581.956,E2 -3581.956} C_VEL
LIN {X 0,Y 544.563,Z 678.885,A -85,B 0,C 180,E1 -3583.505,E2 -3583.505} C_VEL
LIN {X 0,Y 544.561,Z 676.319,A -85,B 0,C 180,E1 -3585.041,E2 -3585.041} C_VEL
LIN {X 0,Y 544.655,Z 672.386,A -85,B 0,C 180,E1 -3586.569,E2 -3586.569} C_VEL
LIN {X 0,Y 544.713,Z 667.208,A -85,B 0,C 180,E1 -3588.086,E2 -3588.086} C_VEL
LIN {X 0,Y 544.812,Z 660.526,A -85,B 0,C 180,E1 -3589.595,E2 -3589.595} C_VEL
LIN {X 0,Y 544.981,Z 652.234,A -85,B 0,C 180,E1 -3591.097,E2 -3591.097} C_VEL
LIN {X 0,Y 545.197,Z 643.518,A -85,B 0,C 180,E1 -3592.407,E2 -3592.407} C_VEL
LIN {X 0,Y 545.357,Z 634.618,A -85,B 0,C 180,E1 -3593.525,E2 -3593.525} C_VEL
LIN {X 0,Y 545.683,Z 624.286,A -85,B 0,C 180,E1 -3594.642,E2 -3594.642} C_VEL
LIN {X 0,Y 545.945,Z 614.067,A -85,B 0,C 180,E1 -3595.57,E2 -3595.57} C_VEL
LIN {X 0,Y 546.28,Z 602.261,A -85,B 0,C 180,E1 -3596.496,E2 -3596.496} C_VEL
LIN {X 0,Y 546.652,Z 589.361,A -85,B 0,C 180,E1 -3597.329,E2 -3597.329} C_VEL
LIN {X 0,Y 546.989,Z 575.337,A -85,B 0,C 180,E1 -3598.067,E2 -3598.067} C_VEL
LIN {X 0,Y 547.285,Z 561.265,A -85,B 0,C 180,E1 -3598.643,E2 -3598.643} C_VEL
LIN {X 0,Y 547.628,Z 545.495,A -85,B 0,C 180,E1 -3599.127,E2 -3599.127} C_VEL
LIN {X 0,Y 547.764,Z 529.171,A -85,B 0,C 180,E1 -3599.448,E2 -3599.448} C_VEL
LIN {X 0,Y 548.46,Z 380.749,A -85,B 0,C 180,E1 -3601.444,E2 -3601.444} C_VEL
LIN {X 0,Y 546.248,Z 370.092,A -85,B 0,C 180,E1 -3601.705,E2 -3601.705} C_VEL
LIN {X 0,Y 546.554,Z 354.287,A -85,B 0,C 180,E1 -3604.055,E2 -3604.055} C_VEL
LIN {X 0,Y 545.192,Z 347.2,A -85,B 0,C 180,E1 -3605.223,E2 -3605.223} C_VEL
LIN {X 0,Y 545.14,Z 347.204,A -85,B 0,C 180,E1 -3607.407,E2 -3607.407} C_VEL
LIN {X 0,Y 545.075,Z 347.216,A -85,B 0,C 180,E1 -3610.399,E2 -3610.399} C_VEL
LIN {X 0,Y 545.084,Z 347.214,A -85,B 0,C 180,E1 -3612.661,E2 -3612.661} C_VEL
LIN {X 0,Y 545.088,Z 347.211,A -85,B 0,C 180,E1 -3614.943,E2 -3614.943} C_VEL
LIN {X 0,Y 545.061,Z 347.215,A -85,B 0,C 180,E1 -3618.026,E2 -3618.026} C_VEL
LIN {X 0,Y 545.094,Z 347.215,A -85,B 0,C 180,E1 -3620.372,E2 -3620.372} C_VEL
LIN {X 0,Y 545.077,Z 347.209,A -85,B 0,C 180,E1 -3623.559,E2 -3623.559} C_VEL
LIN {X 0,Y 545.04,Z 347.218,A -85,B 0,C 180,E1 -3626.002,E2 -3626.002} C_VEL
LIN {X 0,Y 545.024,Z 347.218,A -85,B 0,C 180,E1 -3628.734,E2 -3628.734} C_VEL
LIN {X 0,Y 545.056,Z 347.211,A -85,B 0,C 180,E1 -3631.048,E2 -3631.048} C_VEL
LIN {X 0,Y 545.053,Z 347.214,A -85,B 0,C 180,E1 -3633.673,E2 -3633.673} C_VEL
LIN {X 0,Y 545.001,Z 347.224,A -85,B 0,C 180,E1 -3636.383,E2 -3636.383} C_VEL
LIN {X 0,Y 545.055,Z 347.211,A -85,B 0,C 180,E1 -3639.317,E2 -3639.317} C_VEL
LIN {X 0,Y 545.03,Z 347.222,A -85,B 0,C 180,E1 -3642.107,E2 -3642.107} C_VEL
LIN {X 0,Y 545.013,Z 347.216,A -85,B 0,C 180,E1 -3645.172,E2 -3645.172} C_VEL
LIN {X 0,Y 545.02,Z 347.218,A -85,B 0,C 180,E1 -3648.409,E2 -3648.409} C_VEL
LIN {X 0,Y 545.043,Z 347.213,A -85,B 0,C 180,E1 -3650.814,E2 -3650.814} C_VEL
LIN {X 0,Y 545,Z 347.224,A -85,B 0,C 180,E1 -3653.616,E2 -3653.616} C_VEL
LIN {X 0,Y 545.036,Z 347.22,A -85,B 0,C 180,E1 -3656.325,E2 -3656.325} C_VEL
LIN {X 0,Y 545.041,Z 347.217,A -85,B 0,C 180,E1 -3658.95,E2 -3658.95} C_VEL
LIN {X 0,Y 545.035,Z 347.222,A -85,B 0,C 180,E1 -3661.503,E2 -3661.503} C_VEL
LIN {X 0,Y 545.05,Z 347.305,A -85,B 0,C 180,E1 -3662.755,E2 -3662.755} C_VEL
LIN {X 0,Y 547.234,Z 356.903,A -85,B 0,C 180,E1 -3664.109,E2 -3664.109} C_VEL
LIN {X 0,Y 546.949,Z 374.551,A -85,B 0,C 180,E1 -3666.348,E2 -3666.348} C_VEL
LIN {X 0,Y 546.434,Z 398.682,A -85,B 0,C 180,E1 -3669.354,E2 -3669.354} C_VEL
LIN {X 0,Y 548.484,Z 410.136,A -85,B 0,C 180,E1 -3669.597,E2 -3669.597} C_VEL
LIN {X 0,Y 547.736,Z 565.486,A -85,B 0,C 180,E1 -3671.7,E2 -3671.7} C_VEL
LIN {X 0,Y 547.527,Z 580.669,A -85,B 0,C 180,E1 -3672.057,E2 -3672.057} C_VEL
LIN {X 0,Y 547.229,Z 596.011,A -85,B 0,C 180,E1 -3672.578,E2 -3672.578} C_VEL
LIN {X 0,Y 546.934,Z 609.761,A -85,B 0,C 180,E1 -3673.194,E2 -3673.194} C_VEL
LIN {X 0,Y 546.531,Z 623.238,A -85,B 0,C 180,E1 -3673.949,E2 -3673.949} C_VEL
LIN {X 0,Y 546.151,Z 637.13,A -85,B 0,C 180,E1 -3674.908,E2 -3674.908} C_VEL
LIN {X 0,Y 545.821,Z 649.344,A -85,B 0,C 180,E1 -3675.933,E2 -3675.933} C_VEL
LIN {X 0,Y 545.512,Z 661.5,A -85,B 0,C 180,E1 -3677.159,E2 -3677.159} C_VEL
LIN {X 0,Y 545.176,Z 672.098,A -85,B 0,C 180,E1 -3678.445,E2 -3678.445} C_VEL
LIN {X 0,Y 545.051,Z 681.29,A -85,B 0,C 180,E1 -3679.787,E2 -3679.787} C_VEL
LIN {X 0,Y 544.845,Z 688.744,A -85,B 0,C 180,E1 -3681.094,E2 -3681.094} C_VEL
LIN {X 0,Y 544.746,Z 695.696,A -85,B 0,C 180,E1 -3682.586,E2 -3682.586} C_VEL
LIN {X 0,Y 544.707,Z 701.159,A -85,B 0,C 180,E1 -3684.074,E2 -3684.074} C_VEL
LIN {X 0,Y 544.606,Z 705.289,A -85,B 0,C 180,E1 -3685.558,E2 -3685.558} C_VEL
LIN {X 0,Y 544.644,Z 708.184,A -85,B 0,C 180,E1 -3687.04,E2 -3687.04} C_VEL
LIN {X 0,Y 544.543,Z 709.909,A -85,B 0,C 180,E1 -3688.52,E2 -3688.52} C_VEL
LIN {X 0,Y 544.538,Z 710.5,A -85,B 0,C 180,E1 -3689.999,E2 -3689.999} C_VEL
LIN {X 0,Y 544.543,Z 709.909,A -85,B 0,C 180,E1 -3691.478,E2 -3691.478} C_VEL
LIN {X 0,Y 544.643,Z 708.183,A -85,B 0,C 180,E1 -3692.958,E2 -3692.958} C_VEL
LIN {X 0,Y 544.606,Z 705.292,A -85,B 0,C 180,E1 -3694.44,E2 -3694.44} C_VEL
LIN {X 0,Y 544.708,Z 701.169,A -85,B 0,C 180,E1 -3695.923,E2 -3695.923} C_VEL
LIN {X 0,Y 544.743,Z 695.706,A -85,B 0,C 180,E1 -3697.411,E2 -3697.411} C_VEL
LIN {X 0,Y 544.844,Z 688.751,A -85,B 0,C 180,E1 -3698.903,E2 -3698.903} C_VEL
LIN {X 0,Y 545.073,Z 680.091,A -85,B 0,C 180,E1 -3700.398,E2 -3700.398} C_VEL
LIN {X 0,Y 545.234,Z 670.716,A -85,B 0,C 180,E1 -3701.733,E2 -3701.733} C_VEL
LIN {X 0,Y 545.509,Z 661.519,A -85,B 0,C 180,E1 -3702.839,E2 -3702.839} C_VEL
LIN {X 0,Y 545.826,Z 649.373,A -85,B 0,C 180,E1 -3704.064,E2 -3704.064} C_VEL
LIN {X 0,Y 546.189,Z 636.824,A -85,B 0,C 180,E1 -3705.114,E2 -3705.114} C_VEL
LIN {X 0,Y 546.527,Z 623.273,A -85,B 0,C 180,E1 -3706.049,E2 -3706.049} C_VEL
LIN {X 0,Y 546.972,Z 609.8,A -85,B 0,C 180,E1 -3706.803,E2 -3706.803} C_VEL
LIN {X 0,Y 547.217,Z 596.075,A -85,B 0,C 180,E1 -3707.421,E2 -3707.421} C_VEL
LIN {X 0,Y 547.533,Z 580.763,A -85,B 0,C 180,E1 -3707.941,E2 -3707.941} C_VEL
LIN {X 0,Y 547.716,Z 565.153,A -85,B 0,C 180,E1 -3708.308,E2 -3708.308} C_VEL
LIN {X 0,Y 548.477,Z 410.283,A -85,B 0,C 180,E1 -3710.401,E2 -3710.401} C_VEL
LIN {X 0,Y 547.321,Z 403.246,A -85,B 0,C 180,E1 -3710.54,E2 -3710.54} C_VEL
LIN {X 0,Y 546.479,Z 398.708,A -85,B 0,C 180,E1 -3710.652,E2 -3710.652} C_VEL
LIN {X 0,Y 546.929,Z 376.21,A -85,B 0,C 180,E1 -3713.473,E2 -3713.473} C_VEL
LIN {X 0,Y 547.385,Z 357.303,A -85,B 0,C 180,E1 -3715.881,E2 -3715.881} C_VEL
LIN {X 0,Y 545.038,Z 347.219,A -85,B 0,C 180,E1 -3717.334,E2 -3717.334} C_VEL
LIN {X 0,Y 545.049,Z 347.221,A -85,B 0,C 180,E1 -3720.241,E2 -3720.241} C_VEL
LIN {X 0,Y 545.065,Z 347.211,A -85,B 0,C 180,E1 -3723.06,E2 -3723.06} C_VEL
LIN {X 0,Y 545.01,Z 347.219,A -85,B 0,C 180,E1 -3725.669,E2 -3725.669} C_VEL
LIN {X 0,Y 545.036,Z 347.222,A -85,B 0,C 180,E1 -3728.237,E2 -3728.237} C_VEL
LIN {X 0,Y 545.018,Z 347.215,A -85,B 0,C 180,E1 -3731.118,E2 -3731.118} C_VEL
LIN {X 0,Y 545.026,Z 347.223,A -85,B 0,C 180,E1 -3734.13,E2 -3734.13} C_VEL
LIN {X 0,Y 545.005,Z 347.217,A -85,B 0,C 180,E1 -3736.886,E2 -3736.886} C_VEL
LIN {X 0,Y 545.046,Z 347.216,A -85,B 0,C 180,E1 -3739.856,E2 -3739.856} C_VEL
LIN {X 0,Y 545.004,Z 347.218,A -85,B 0,C 180,E1 -3742.694,E2 -3742.694} C_VEL
LIN {X 0,Y 545.044,Z 347.213,A -85,B 0,C 180,E1 -3745.61,E2 -3745.61} C_VEL
LIN {X 0,Y 545.044,Z 347.218,A -85,B 0,C 180,E1 -3748.321,E2 -3748.321} C_VEL
LIN {X 0,Y 545.008,Z 347.218,A -85,B 0,C 180,E1 -3750.658,E2 -3750.658} C_VEL
LIN {X 0,Y 545.028,Z 347.213,A -85,B 0,C 180,E1 -3753.172,E2 -3753.172} C_VEL
LIN {X 0,Y 545.032,Z 347.22,A -85,B 0,C 180,E1 -3756.275,E2 -3756.275} C_VEL
LIN {X 0,Y 545.034,Z 347.213,A -85,B 0,C 180,E1 -3758.836,E2 -3758.836} C_VEL
LIN {X 0,Y 545.032,Z 347.213,A -85,B 0,C 180,E1 -3761.194,E2 -3761.194} C_VEL
LIN {X 0,Y 545.02,Z 347.22,A -85,B 0,C 180,E1 -3764.289,E2 -3764.289} C_VEL
LIN {X 0,Y 545.039,Z 347.214,A -85,B 0,C 180,E1 -3766.579,E2 -3766.579} C_VEL
LIN {X 0,Y 545.099,Z 347.205,A -85,B 0,C 180,E1 -3768.849,E2 -3768.849} C_VEL
LIN {X 0,Y 545.066,Z 347.215,A -85,B 0,C 180,E1 -3771.846,E2 -3771.846} C_VEL
LIN {X 0,Y 545.149,Z 347.198,A -85,B 0,C 180,E1 -3774.823,E2 -3774.823} C_VEL
LIN {X 0,Y 545.177,Z 347.201,A -85,B 0,C 180,E1 -3777.784,E2 -3777.784} C_VEL
LIN {X 0,Y 545.176,Z 347.205,A -85,B 0,C 180,E1 -3780,E2 -3780} C_VEL
LIN {X 0,Y 545.126,Z 347.201,A -85,B 0,C 180,E1 -3782.956,E2 -3782.956} C_VEL
LIN {X 0,Y 545.113,Z 347.212,A -85,B 0,C 180,E1 -3785.92,E2 -3785.92} C_VEL
LIN {X 0,Y 545.075,Z 347.207,A -85,B 0,C 180,E1 -3788.901,E2 -3788.901} C_VEL
LIN {X 0,Y 545.051,Z 347.22,A -85,B 0,C 180,E1 -3791.906,E2 -3791.906} C_VEL
LIN {X 0,Y 545.064,Z 347.209,A -85,B 0,C 180,E1 -3794.944,E2 -3794.944} C_VEL
LIN {X 0,Y 545.034,Z 347.221,A -85,B 0,C 180,E1 -3798.028,E2 -3798.028} C_VEL
LIN {X 0,Y 545.069,Z 347.211,A -85,B 0,C 180,E1 -3800.373,E2 -3800.373} C_VEL
LIN {X 0,Y 545.058,Z 347.214,A -85,B 0,C 180,E1 -3803.561,E2 -3803.561} C_VEL
LIN {X 0,Y 545.022,Z 347.222,A -85,B 0,C 180,E1 -3806.004,E2 -3806.004} C_VEL
LIN {X 0,Y 545.008,Z 347.216,A -85,B 0,C 180,E1 -3808.736,E2 -3808.736} C_VEL
LIN {X 0,Y 545.049,Z 347.211,A -85,B 0,C 180,E1 -3811.049,E2 -3811.049} C_VEL
LIN {X 0,Y 545.045,Z 347.217,A -85,B 0,C 180,E1 -3813.756,E2 -3813.756} C_VEL
LIN {X 0,Y 545.004,Z 347.216,A -85,B 0,C 180,E1 -3816.92,E2 -3816.92} C_VEL
LIN {X 0,Y 545.003,Z 347.216,A -85,B 0,C 180,E1 -3816.973,E2 -3816.973} C_VEL
LIN {X 0,Y 544.337,Z 347.306,A -85,B 0,C 180,E1 -3817.59,E2 -3817.59} C_VEL
LIN {X 0,Y 541.492,Z 347.661,A -85,B 0,C 180,E1 -3818.591,E2 -3818.591} C_VEL
LIN {X 0,Y 539.089,Z 347.961,A -85,B 0,C 180,E1 -3819.398,E2 -3819.398} C_VEL
LIN {X 0,Y 538.059,Z 348.088,A -85,B 0,C 180,E1 -3820.02,E2 -3820.02} C_VEL
LIN {X 0,Y 537.975,Z 348.094,A -85,B 0,C 180,E1 -3820.231,E2 -3820.231} C_VEL
LIN {X 0,Y 537.961,Z 348.094,A -85,B 0,C 180,E1 -3822.982,E2 -3822.982} C_VEL
LIN {X 0,Y 538.001,Z 348.097,A -85,B 0,C 180,E1 -3825.929,E2 -3825.929} C_VEL
LIN {X 0,Y 537.994,Z 348.091,A -85,B 0,C 180,E1 -3829.26,E2 -3829.26} C_VEL
LIN {X 0,Y 537.978,Z 348.096,A -85,B 0,C 180,E1 -3832.123,E2 -3832.123} C_VEL
LIN {X 0,Y 537.982,Z 348.091,A -85,B 0,C 180,E1 -3834.916,E2 -3834.916} C_VEL
LIN {X 0,Y 538.011,Z 348.094,A -85,B 0,C 180,E1 -3837.619,E2 -3837.619} C_VEL
LIN {X 0,Y 537.993,Z 348.092,A -85,B 0,C 180,E1 -3840.239,E2 -3840.239} C_VEL
LIN {X 0,Y 537.992,Z 348.09,A -85,B 0,C 180,E1 -3842.794,E2 -3842.794} C_VEL
LIN {X 0,Y 537.982,Z 348.094,A -85,B 0,C 180,E1 -3845.291,E2 -3845.291} C_VEL
LIN {X 0,Y 538.014,Z 348.092,A -85,B 0,C 180,E1 -3848.044,E2 -3848.044} C_VEL
LIN {X 0,Y 538.08,Z 348.082,A -85,B 0,C 180,E1 -3850.149,E2 -3850.149} C_VEL
LIN {X 0,Y 537.985,Z 348.094,A -85,B 0,C 180,E1 -3853.299,E2 -3853.299} C_VEL
LIN {X 0,Y 538.051,Z 348.091,A -85,B 0,C 180,E1 -3855.632,E2 -3855.632} C_VEL
LIN {X 0,Y 538.077,Z 348.079,A -85,B 0,C 180,E1 -3858.703,E2 -3858.703} C_VEL
LIN {X 0,Y 538.042,Z 348.093,A -85,B 0,C 180,E1 -3861.74,E2 -3861.74} C_VEL
LIN {X 0,Y 538.129,Z 348.073,A -85,B 0,C 180,E1 -3864.756,E2 -3864.756} C_VEL
LIN {X 0,Y 538.165,Z 348.076,A -85,B 0,C 180,E1 -3867.756,E2 -3867.756} C_VEL
LIN {X 0,Y 538.163,Z 348.073,A -85,B 0,C 180,E1 -3870.001,E2 -3870.001} C_VEL
LIN {X 0,Y 538.12,Z 348.075,A -85,B 0,C 180,E1 -3872.996,E2 -3872.996} C_VEL
LIN {X 0,Y 538.093,Z 348.081,A -85,B 0,C 180,E1 -3875.999,E2 -3875.999} C_VEL
LIN {X 0,Y 538.051,Z 348.084,A -85,B 0,C 180,E1 -3879.019,E2 -3879.019} C_VEL
LIN {X 0,Y 538.06,Z 348.084,A -85,B 0,C 180,E1 -3882.064,E2 -3882.064} C_VEL
LIN {X 0,Y 538.044,Z 348.086,A -85,B 0,C 180,E1 -3885.145,E2 -3885.145} C_VEL
LIN {X 0,Y 538.009,Z 348.089,A -85,B 0,C 180,E1 -3888.272,E2 -3888.272} C_VEL
LIN {X 0,Y 538.041,Z 348.084,A -85,B 0,C 180,E1 -3890.652,E2 -3890.652} C_VEL
LIN {X 0,Y 538.013,Z 348.092,A -85,B 0,C 180,E1 -3893.878,E2 -3893.878} C_VEL
LIN {X 0,Y 537.995,Z 348.09,A -85,B 0,C 180,E1 -3896.37,E2 -3896.37} C_VEL
LIN {X 0,Y 537.998,Z 348.09,A -85,B 0,C 180,E1 -3898.926,E2 -3898.926} C_VEL
LIN {X 0,Y 538.016,Z 348.091,A -85,B 0,C 180,E1 -3901.887,E2 -3901.887} C_VEL
LIN {X 0,Y 538.006,Z 348.088,A -85,B 0,C 180,E1 -3904.616,E2 -3904.616} C_VEL
LIN {X 0,Y 538.005,Z 348.095,A -85,B 0,C 180,E1 -3907.169,E2 -3907.169} C_VEL
LIN {X 0,Y 538.026,Z 348.093,A -85,B 0,C 180,E1 -3909.798,E2 -3909.798} C_VEL
LIN {X 0,Y 538.005,Z 348.092,A -85,B 0,C 180,E1 -3912.788,E2 -3912.788} C_VEL
LIN {X 0,Y 538.001,Z 348.096,A -85,B 0,C 180,E1 -3915.137,E2 -3915.137} C_VEL
LIN {X 0,Y 538.051,Z 348.16,A -85,B 0,C 180,E1 -3916.73,E2 -3916.73} C_VEL
LIN {X 0,Y 539.629,Z 356.356,A -85,B 0,C 180,E1 -3918.049,E2 -3918.049} C_VEL
LIN {X 0,Y 539.368,Z 370.191,A -85,B 0,C 180,E1 -3920.12,E2 -3920.12} C_VEL
LIN {X 0,Y 541.815,Z 381.643,A -85,B 0,C 180,E1 -3920.397,E2 -3920.397} C_VEL
LIN {X 0,Y 541.017,Z 534.671,A -85,B 0,C 180,E1 -3922.508,E2 -3922.508} C_VEL
LIN {X 0,Y 540.709,Z 550.991,A -85,B 0,C 180,E1 -3922.887,E2 -3922.887} C_VEL
LIN {X 0,Y 540.42,Z 565.569,A -85,B 0,C 180,E1 -3923.387,E2 -3923.387} C_VEL
LIN {X 0,Y 540.073,Z 578.213,A -85,B 0,C 180,E1 -3923.952,E2 -3923.952} C_VEL
LIN {X 0,Y 539.78,Z 589.91,A -85,B 0,C 180,E1 -3924.592,E2 -3924.592} C_VEL
LIN {X 0,Y 539.385,Z 601.831,A -85,B 0,C 180,E1 -3925.36,E2 -3925.36} C_VEL
LIN {X 0,Y 539.048,Z 614.787,A -85,B 0,C 180,E1 -3926.386,E2 -3926.386} C_VEL
LIN {X 0,Y 538.646,Z 626.946,A -85,B 0,C 180,E1 -3927.549,E2 -3927.549} C_VEL
LIN {X 0,Y 538.339,Z 637.472,A -85,B 0,C 180,E1 -3928.739,E2 -3928.739} C_VEL
LIN {X 0,Y 538.096,Z 646.915,A -85,B 0,C 180,E1 -3930.028,E2 -3930.028} C_VEL
LIN {X 0,Y 537.896,Z 654.876,A -85,B 0,C 180,E1 -3931.303,E2 -3931.303} C_VEL
LIN {X 0,Y 537.708,Z 662.377,A -85,B 0,C 180,E1 -3932.776,E2 -3932.776} C_VEL
LIN {X 0,Y 537.638,Z 667.665,A -85,B 0,C 180,E1 -3934.029,E2 -3934.029} C_VEL
LIN {X 0,Y 537.567,Z 671.861,A -85,B 0,C 180,E1 -3935.269,E2 -3935.269} C_VEL
LIN {X 0,Y 537.51,Z 676.121,A -85,B 0,C 180,E1 -3936.905,E2 -3936.905} C_VEL
LIN {X 0,Y 537.472,Z 678.839,A -85,B 0,C 180,E1 -3938.523,E2 -3938.523} C_VEL
LIN {X 0,Y 537.463,Z 680.277,A -85,B 0,C 180,E1 -3940.124,E2 -3940.124} C_VEL
LIN {X 0,Y 537.448,Z 680.344,A -85,B 0,C 180,E1 -3941.709,E2 -3941.709} C_VEL
LIN {X 0,Y 537.46,Z 679.215,A -85,B 0,C 180,E1 -3943.281,E2 -3943.281} C_VEL
LIN {X 0,Y 537.454,Z 676.8,A -85,B 0,C 180,E1 -3944.839,E2 -3944.839} C_VEL
LIN {X 0,Y 537.553,Z 673.125,A -85,B 0,C 180,E1 -3946.389,E2 -3946.389} C_VEL
LIN {X 0,Y 537.616,Z 668.156,A -85,B 0,C 180,E1 -3947.927,E2 -3947.927} C_VEL
LIN {X 0,Y 537.711,Z 661.71,A -85,B 0,C 180,E1 -3949.456,E2 -3949.456} C_VEL
LIN {X 0,Y 537.894,Z 653.754,A -85,B 0,C 180,E1 -3950.979,E2 -3950.979} C_VEL
LIN {X 0,Y 538.133,Z 645.255,A -85,B 0,C 180,E1 -3952.307,E2 -3952.307} C_VEL
LIN {X 0,Y 538.363,Z 635.131,A -85,B 0,C 180,E1 -3953.629,E2 -3953.629} C_VEL
LIN {X 0,Y 538.693,Z 624.879,A -85,B 0,C 180,E1 -3954.76,E2 -3954.76} C_VEL
LIN {X 0,Y 539.021,Z 613.662,A -85,B 0,C 180,E1 -3955.794,E2 -3955.794} C_VEL
LIN {X 0,Y 539.414,Z 601.786,A -85,B 0,C 180,E1 -3956.732,E2 -3956.732} C_VEL
LIN {X 0,Y 539.822,Z 588.732,A -85,B 0,C 180,E1 -3957.575,E2 -3957.575} C_VEL
LIN {X 0,Y 540.204,Z 574.466,A -85,B 0,C 180,E1 -3958.322,E2 -3958.322} C_VEL
LIN {X 0,Y 540.486,Z 559.997,A -85,B 0,C 180,E1 -3958.905,E2 -3958.905} C_VEL
LIN {X 0,Y 540.843,Z 545.397,A -85,B 0,C 180,E1 -3959.348,E2 -3959.348} C_VEL
LIN {X 0,Y 541.006,Z 530.279,A -85,B 0,C 180,E1 -3959.651,E2 -3959.651} C_VEL
LIN {X 0,Y 541.752,Z 381.192,A -85,B 0,C 180,E1 -3961.703,E2 -3961.703} C_VEL
LIN {X 0,Y 539.415,Z 370.484,A -85,B 0,C 180,E1 -3961.96,E2 -3961.96} C_VEL
LIN {X 0,Y 539.731,Z 356.208,A -85,B 0,C 180,E1 -3964.107,E2 -3964.107} C_VEL
LIN {X 0,Y 538.14,Z 348.078,A -85,B 0,C 180,E1 -3965.456,E2 -3965.456} C_VEL
LIN {X 0,Y 538.063,Z 348.09,A -85,B 0,C 180,E1 -3968.261,E2 -3968.261} C_VEL
LIN {X 0,Y 538.09,Z 348.079,A -85,B 0,C 180,E1 -3971.598,E2 -3971.598} C_VEL
LIN {X 0,Y 538.064,Z 348.087,A -85,B 0,C 180,E1 -3974.857,E2 -3974.857} C_VEL
LIN {X 0,Y 538.041,Z 348.086,A -85,B 0,C 180,E1 -3977.532,E2 -3977.532} C_VEL
LIN {X 0,Y 538.04,Z 348.09,A -85,B 0,C 180,E1 -3980.651,E2 -3980.651} C_VEL
LIN {X 0,Y 538.01,Z 348.092,A -85,B 0,C 180,E1 -3983.877,E2 -3983.877} C_VEL
LIN {X 0,Y 537.984,Z 348.1,A -85,B 0,C 180,E1 -3986.37,E2 -3986.37} C_VEL
LIN {X 0,Y 537.995,Z 348.092,A -85,B 0,C 180,E1 -3988.925,E2 -3988.925} C_VEL
LIN {X 0,Y 538,Z 348.094,A -85,B 0,C 180,E1 -3991.884,E2 -3991.884} C_VEL
LIN {X 0,Y 537.997,Z 348.094,A -85,B 0,C 180,E1 -3994.614,E2 -3994.614} C_VEL
LIN {X 0,Y 537.98,Z 348.098,A -85,B 0,C 180,E1 -3997.879,E2 -3997.879} C_VEL
LIN {X 0,Y 537.96,Z 348.096,A -85,B 0,C 180,E1 -4000.784,E2 -4000.784} C_VEL
LIN {X 0,Y 537.979,Z 348.098,A -85,B 0,C 180,E1 -4003.818,E2 -4003.818} C_VEL
LIN {X 0,Y 537.979,Z 348.099,A -85,B 0,C 180,E1 -4006.181,E2 -4006.181} C_VEL
LIN {X 0,Y 537.953,Z 348.096,A -85,B 0,C 180,E1 -4009.264,E2 -4009.264} C_VEL
LIN {X 0,Y 537.971,Z 348.1,A -85,B 0,C 180,E1 -4012.12,E2 -4012.12} C_VEL
LIN {X 0,Y 537.992,Z 348.096,A -85,B 0,C 180,E1 -4015.385,E2 -4015.385} C_VEL
LIN {X 0,Y 537.997,Z 348.1,A -85,B 0,C 180,E1 -4018.115,E2 -4018.115} C_VEL
LIN {X 0,Y 537.986,Z 348.097,A -85,B 0,C 180,E1 -4021.095,E2 -4021.095} C_VEL
LIN {X 0,Y 537.984,Z 348.165,A -85,B 0,C 180,E1 -4022.513,E2 -4022.513} C_VEL
LIN {X 0,Y 540.4,Z 358.618,A -85,B 0,C 180,E1 -4024.013,E2 -4024.013} C_VEL
LIN {X 0,Y 540.085,Z 375.693,A -85,B 0,C 180,E1 -4026.208,E2 -4026.208} C_VEL
LIN {X 0,Y 539.554,Z 398.406,A -85,B 0,C 180,E1 -4029.079,E2 -4029.079} C_VEL
LIN {X 0,Y 541.786,Z 410.216,A -85,B 0,C 180,E1 -4029.345,E2 -4029.345} C_VEL
LIN {X 0,Y 540.96,Z 565.163,A -85,B 0,C 180,E1 -4031.474,E2 -4031.474} C_VEL
LIN {X 0,Y 540.73,Z 580.947,A -85,B 0,C 180,E1 -4031.848,E2 -4031.848} C_VEL
LIN {X 0,Y 540.411,Z 595.733,A -85,B 0,C 180,E1 -4032.351,E2 -4032.351} C_VEL
LIN {X 0,Y 540.105,Z 609.666,A -85,B 0,C 180,E1 -4032.975,E2 -4032.975} C_VEL
LIN {X 0,Y 539.663,Z 623.236,A -85,B 0,C 180,E1 -4033.739,E2 -4033.739} C_VEL
LIN {X 0,Y 539.323,Z 636.232,A -85,B 0,C 180,E1 -4034.645,E2 -4034.645} C_VEL
LIN {X 0,Y 538.901,Z 648.277,A -85,B 0,C 180,E1 -4035.652,E2 -4035.652} C_VEL
LIN {X 0,Y 538.594,Z 659.738,A -85,B 0,C 180,E1 -4036.799,E2 -4036.799} C_VEL
LIN {X 0,Y 538.284,Z 669.38,A -85,B 0,C 180,E1 -4037.941,E2 -4037.941} C_VEL
LIN {X 0,Y 538.064,Z 678.847,A -85,B 0,C 180,E1 -4039.272,E2 -4039.272} C_VEL
LIN {X 0,Y 537.825,Z 686.729,A -85,B 0,C 180,E1 -4040.598,E2 -4040.598} C_VEL
LIN {X 0,Y 537.7,Z 694.085,A -85,B 0,C 180,E1 -4042.111,E2 -4042.111} C_VEL
LIN {X 0,Y 537.623,Z 699.401,A -85,B 0,C 180,E1 -4043.462,E2 -4043.462} C_VEL
LIN {X 0,Y 537.574,Z 703.383,A -85,B 0,C 180,E1 -4044.748,E2 -4044.748} C_VEL
LIN {X 0,Y 537.562,Z 706.885,A -85,B 0,C 180,E1 -4046.251,E2 -4046.251} C_VEL
LIN {X 0,Y 537.487,Z 709.188,A -85,B 0,C 180,E1 -4047.751,E2 -4047.751} C_VEL
LIN {X 0,Y 537.438,Z 710.348,A -85,B 0,C 180,E1 -4049.25,E2 -4049.25} C_VEL
LIN {X 0,Y 537.438,Z 710.347,A -85,B 0,C 180,E1 -4050.748,E2 -4050.748} C_VEL
LIN {X 0,Y 537.487,Z 709.188,A -85,B 0,C 180,E1 -4052.247,E2 -4052.247} C_VEL
LIN {X 0,Y 537.562,Z 706.886,A -85,B 0,C 180,E1 -4053.747,E2 -4053.747} C_VEL
LIN {X 0,Y 537.574,Z 703.39,A -85,B 0,C 180,E1 -4055.25,E2 -4055.25} C_VEL
LIN {X 0,Y 537.662,Z 698.614,A -85,B 0,C 180,E1 -4056.755,E2 -4056.755} C_VEL
LIN {X 0,Y 537.733,Z 692.426,A -85,B 0,C 180,E1 -4058.265,E2 -4058.265} C_VEL
LIN {X 0,Y 537.859,Z 684.65,A -85,B 0,C 180,E1 -4059.779,E2 -4059.779} C_VEL
LIN {X 0,Y 538.1,Z 676.375,A -85,B 0,C 180,E1 -4061.106,E2 -4061.106} C_VEL
LIN {X 0,Y 538.356,Z 666.402,A -85,B 0,C 180,E1 -4062.438,E2 -4062.438} C_VEL
LIN {X 0,Y 538.661,Z 656.196,A -85,B 0,C 180,E1 -4063.581,E2 -4063.581} C_VEL
LIN {X 0,Y 539.026,Z 644.033,A -85,B 0,C 180,E1 -4064.728,E2 -4064.728} C_VEL
LIN {X 0,Y 539.461,Z 631.841,A -85,B 0,C 180,E1 -4065.681,E2 -4065.681} C_VEL
LIN {X 0,Y 539.832,Z 618.516,A -85,B 0,C 180,E1 -4066.545,E2 -4066.545} C_VEL
LIN {X 0,Y 540.214,Z 603.71,A -85,B 0,C 180,E1 -4067.312,E2 -4067.312} C_VEL
LIN {X 0,Y 540.569,Z 589.366,A -85,B 0,C 180,E1 -4067.886,E2 -4067.886} C_VEL
LIN {X 0,Y 540.813,Z 574.396,A -85,B 0,C 180,E1 -4068.33,E2 -4068.33} C_VEL
LIN {X 0,Y 541.009,Z 559.126,A -85,B 0,C 180,E1 -4068.628,E2 -4068.628} C_VEL
LIN {X 0,Y 541.783,Z 410.317,A -85,B 0,C 180,E1 -4070.653,E2 -4070.653} C_VEL
LIN {X 0,Y 539.566,Z 398.554,A -85,B 0,C 180,E1 -4070.929,E2 -4070.929} C_VEL
LIN {X 0,Y 540.064,Z 377.639,A -85,B 0,C 180,E1 -4073.587,E2 -4073.587} C_VEL
LIN {X 0,Y 540.545,Z 358.916,A -85,B 0,C 180,E1 -4076.002,E2 -4076.002} C_VEL
LIN {X 0,Y 538.015,Z 348.095,A -85,B 0,C 180,E1 -4077.583,E2 -4077.583} C_VEL
LIN {X 0,Y 538.005,Z 348.095,A -85,B 0,C 180,E1 -4080.626,E2 -4080.626} C_VEL
LIN {X 0,Y 538.011,Z 348.089,A -85,B 0,C 180,E1 -4083.277,E2 -4083.277} C_VEL
LIN {X 0,Y 537.977,Z 348.099,A -85,B 0,C 180,E1 -4086.004,E2 -4086.004} C_VEL
LIN {X 0,Y 537.998,Z 348.091,A -85,B 0,C 180,E1 -4088.83,E2 -4088.83} C_VEL
LIN {X 0,Y 537.988,Z 348.095,A -85,B 0,C 180,E1 -4091.874,E2 -4091.874} C_VEL
LIN {X 0,Y 537.981,Z 348.092,A -85,B 0,C 180,E1 -4094.863,E2 -4094.863} C_VEL
LIN {X 0,Y 537.96,Z 348.094,A -85,B 0,C 180,E1 -4097.208,E2 -4097.208} C_VEL
LIN {X 0,Y 537.994,Z 348.099,A -85,B 0,C 180,E1 -4100.201,E2 -4100.201} C_VEL
LIN {X 0,Y 537.957,Z 348.094,A -85,B 0,C 180,E1 -4103.062,E2 -4103.062} C_VEL
LIN {X 0,Y 537.992,Z 348.094,A -85,B 0,C 180,E1 -4105.825,E2 -4105.825} C_VEL
LIN {X 0,Y 537.993,Z 348.094,A -85,B 0,C 180,E1 -4108.498,E2 -4108.498} C_VEL
LIN {X 0,Y 537.969,Z 348.093,A -85,B 0,C 180,E1 -4111.095,E2 -4111.095} C_VEL
LIN {X 0,Y 537.967,Z 348.095,A -85,B 0,C 180,E1 -4113.63,E2 -4113.63} C_VEL
LIN {X 0,Y 537.991,Z 348.099,A -85,B 0,C 180,E1 -4116.122,E2 -4116.122} C_VEL
LIN {X 0,Y 537.999,Z 348.092,A -85,B 0,C 180,E1 -4118.545,E2 -4118.545} C_VEL
LIN {X 0,Y 537.998,Z 348.089,A -85,B 0,C 180,E1 -4120.939,E2 -4120.939} C_VEL
LIN {X 0,Y 537.953,Z 348.095,A -85,B 0,C 180,E1 -4123.297,E2 -4123.297} C_VEL
LIN {X 0,Y 538.033,Z 348.088,A -85,B 0,C 180,E1 -4125.63,E2 -4125.63} C_VEL
LIN {X 0,Y 538.059,Z 348.083,A -85,B 0,C 180,E1 -4128.701,E2 -4128.701} C_VEL
LIN {X 0,Y 538.033,Z 348.09,A -85,B 0,C 180,E1 -4131.739,E2 -4131.739} C_VEL
LIN {X 0,Y 538.111,Z 348.076,A -85,B 0,C 180,E1 -4134.755,E2 -4134.755} C_VEL
LIN {X 0,Y 538.148,Z 348.076,A -85,B 0,C 180,E1 -4137.755,E2 -4137.755} C_VEL
LIN {X 0,Y 538.144,Z 348.081,A -85,B 0,C 180,E1 -4140,E2 -4140} C_VEL
LIN {X 0,Y 538.094,Z 348.077,A -85,B 0,C 180,E1 -4142.995,E2 -4142.995} C_VEL
LIN {X 0,Y 538.07,Z 348.09,A -85,B 0,C 180,E1 -4145.998,E2 -4145.998} C_VEL
LIN {X 0,Y 538.028,Z 348.085,A -85,B 0,C 180,E1 -4149.019,E2 -4149.019} C_VEL
LIN {X 0,Y 538.022,Z 348.094,A -85,B 0,C 180,E1 -4152.064,E2 -4152.064} C_VEL
LIN {X 0,Y 538.023,Z 348.086,A -85,B 0,C 180,E1 -4155.145,E2 -4155.145} C_VEL
LIN {X 0,Y 537.989,Z 348.095,A -85,B 0,C 180,E1 -4158.272,E2 -4158.272} C_VEL
LIN {X 0,Y 538.013,Z 348.088,A -85,B 0,C 180,E1 -4160.653,E2 -4160.653} C_VEL
LIN {X 0,Y 537.992,Z 348.09,A -85,B 0,C 180,E1 -4163.073,E2 -4163.073} C_VEL
LIN {X 0,Y 537.976,Z 348.097,A -85,B 0,C 180,E1 -4165.661,E2 -4165.661} C_VEL
LIN {X 0,Y 537.96,Z 348.101,A -85,B 0,C 180,E1 -4168.055,E2 -4168.055} C_VEL
LIN {X 0,Y 537.992,Z 348.09,A -85,B 0,C 180,E1 -4170.629,E2 -4170.629} C_VEL
LIN {X 0,Y 538.034,Z 348.086,A -85,B 0,C 180,E1 -4173.284,E2 -4173.284} C_VEL
LIN {X 0,Y 537.95,Z 348.102,A -85,B 0,C 180,E1 -4176.008,E2 -4176.008} C_VEL
LIN {X 0,Y 537.997,Z 348.089,A -85,B 0,C 180,E1 -4178.832,E2 -4178.832} C_VEL
LIN {X 0,Y 537.975,Z 348.094,A -85,B 0,C 180,E1 -4180.231,E2 -4180.231} C_VEL
LIN {X 0,Y 537.31,Z 348.176,A -85,B 0,C 180,E1 -4180.856,E2 -4180.856} C_VEL
LIN {X 0,Y 534.456,Z 348.54,A -85,B 0,C 180,E1 -4181.871,E2 -4181.871} C_VEL
LIN {X 0,Y 532.04,Z 348.841,A -85,B 0,C 180,E1 -4182.687,E2 -4182.687} C_VEL
LIN {X 0,Y 531.001,Z 348.967,A -85,B 0,C 180,E1 -4183.318,E2 -4183.318} C_VEL
LIN {X 0,Y 530.916,Z 348.975,A -85,B 0,C 180,E1 -4183.532,E2 -4183.532} C_VEL
LIN {X 0,Y 530.928,Z 348.971,A -85,B 0,C 180,E1 -4186.504,E2 -4186.504} C_VEL
LIN {X 0,Y 530.939,Z 348.974,A -85,B 0,C 180,E1 -4189.565,E2 -4189.565} C_VEL
LIN {X 0,Y 530.931,Z 348.97,A -85,B 0,C 180,E1 -4192.583,E2 -4192.583} C_VEL
LIN {X 0,Y 530.968,Z 348.967,A -85,B 0,C 180,E1 -4195.31,E2 -4195.31} C_VEL
LIN {X 0,Y 530.961,Z 348.971,A -85,B 0,C 180,E1 -4198.033,E2 -4198.033} C_VEL
LIN {X 0,Y 530.959,Z 348.966,A -85,B 0,C 180,E1 -4200.881,E2 -4200.881} C_VEL
LIN {X 0,Y 530.944,Z 348.97,A -85,B 0,C 180,E1 -4203.255,E2 -4203.255} C_VEL
LIN {X 0,Y 530.951,Z 348.973,A -85,B 0,C 180,E1 -4205.97,E2 -4205.97} C_VEL
LIN {X 0,Y 530.996,Z 348.962,A -85,B 0,C 180,E1 -4209.063,E2 -4209.063} C_VEL
LIN {X 0,Y 530.969,Z 348.97,A -85,B 0,C 180,E1 -4211.479,E2 -4211.479} C_VEL
LIN {X 0,Y 530.984,Z 348.963,A -85,B 0,C 180,E1 -4214.651,E2 -4214.651} C_VEL
LIN {X 0,Y 531.025,Z 348.966,A -85,B 0,C 180,E1 -4217.776,E2 -4217.776} C_VEL
LIN {X 0,Y 530.973,Z 348.968,A -85,B 0,C 180,E1 -4220.093,E2 -4220.093} C_VEL
LIN {X 0,Y 531.014,Z 348.961,A -85,B 0,C 180,E1 -4223.16,E2 -4223.16} C_VEL
LIN {X 0,Y 530.987,Z 348.968,A -85,B 0,C 180,E1 -4225.446,E2 -4225.446} C_VEL
LIN {X 0,Y 531.137,Z 348.952,A -85,B 0,C 180,E1 -4227.726,E2 -4227.726} C_VEL
LIN {X 0,Y 531.131,Z 348.949,A -85,B 0,C 180,E1 -4230.001,E2 -4230.001} C_VEL
LIN {X 0,Y 531.062,Z 348.955,A -85,B 0,C 180,E1 -4233.035,E2 -4233.035} C_VEL
LIN {X 0,Y 531.052,Z 348.957,A -85,B 0,C 180,E1 -4236.079,E2 -4236.079} C_VEL
LIN {X 0,Y 531.014,Z 348.962,A -85,B 0,C 180,E1 -4239.139,E2 -4239.139} C_VEL
LIN {X 0,Y 531.054,Z 348.963,A -85,B 0,C 180,E1 -4241.671,E2 -4241.671} C_VEL
LIN {X 0,Y 531.035,Z 348.958,A -85,B 0,C 180,E1 -4244.955,E2 -4244.955} C_VEL
LIN {X 0,Y 530.973,Z 348.964,A -85,B 0,C 180,E1 -4248.523,E2 -4248.523} C_VEL
LIN {X 0,Y 531.003,Z 348.962,A -85,B 0,C 180,E1 -4250.939,E2 -4250.939} C_VEL
LIN {X 0,Y 530.957,Z 348.967,A -85,B 0,C 180,E1 -4254.227,E2 -4254.227} C_VEL
LIN {X 0,Y 530.962,Z 348.966,A -85,B 0,C 180,E1 -4256.747,E2 -4256.747} C_VEL
LIN {X 0,Y 530.968,Z 348.971,A -85,B 0,C 180,E1 -4259.324,E2 -4259.324} C_VEL
LIN {X 0,Y 530.971,Z 348.966,A -85,B 0,C 180,E1 -4262.1,E2 -4262.1} C_VEL
LIN {X 0,Y 530.966,Z 348.966,A -85,B 0,C 180,E1 -4264.85,E2 -4264.85} C_VEL
LIN {X 0,Y 530.969,Z 348.975,A -85,B 0,C 180,E1 -4267.508,E2 -4267.508} C_VEL
LIN {X 0,Y 530.971,Z 348.967,A -85,B 0,C 180,E1 -4270.435,E2 -4270.435} C_VEL
LIN {X 0,Y 530.949,Z 348.975,A -85,B 0,C 180,E1 -4273.279,E2 -4273.279} C_VEL
LIN {X 0,Y 530.97,Z 348.973,A -85,B 0,C 180,E1 -4276.244,E2 -4276.244} C_VEL
LIN {X 0,Y 531.003,Z 349.08,A -85,B 0,C 180,E1 -4276.509,E2 -4276.509} C_VEL
LIN {X 0,Y 532.583,Z 356.302,A -85,B 0,C 180,E1 -4277.701,E2 -4277.701} C_VEL
LIN {X 0,Y 532.659,Z 364.738,A -85,B 0,C 180,E1 -4278.991,E2 -4278.991} C_VEL
LIN {X 0,Y 532.507,Z 370.349,A -85,B 0,C 180,E1 -4279.835,E2 -4279.835} C_VEL
LIN {X 0,Y 535.143,Z 383.413,A -85,B 0,C 180,E1 -4280.154,E2 -4280.154} C_VEL
LIN {X 0,Y 534.206,Z 535.317,A -85,B 0,C 180,E1 -4282.288,E2 -4282.288} C_VEL
LIN {X 0,Y 533.944,Z 551.051,A -85,B 0,C 180,E1 -4282.663,E2 -4282.663} C_VEL
LIN {X 0,Y 533.605,Z 565.009,A -85,B 0,C 180,E1 -4283.14,E2 -4283.14} C_VEL
LIN {X 0,Y 533.268,Z 578.38,A -85,B 0,C 180,E1 -4283.742,E2 -4283.742} C_VEL
LIN {X 0,Y 532.899,Z 590.47,A -85,B 0,C 180,E1 -4284.413,E2 -4284.413} C_VEL
LIN {X 0,Y 532.456,Z 603.02,A -85,B 0,C 180,E1 -4285.244,E2 -4285.244} C_VEL
LIN {X 0,Y 532.089,Z 616.23,A -85,B 0,C 180,E1 -4286.319,E2 -4286.319} C_VEL
LIN {X 0,Y 531.69,Z 626.907,A -85,B 0,C 180,E1 -4287.363,E2 -4287.363} C_VEL
LIN {X 0,Y 531.354,Z 636.898,A -85,B 0,C 180,E1 -4288.503,E2 -4288.503} C_VEL
LIN {X 0,Y 531.071,Z 646.435,A -85,B 0,C 180,E1 -4289.809,E2 -4289.809} C_VEL
LIN {X 0,Y 530.827,Z 655.109,A -85,B 0,C 180,E1 -4291.217,E2 -4291.217} C_VEL
LIN {X 0,Y 530.661,Z 661.798,A -85,B 0,C 180,E1 -4292.542,E2 -4292.542} C_VEL
LIN {X 0,Y 530.557,Z 668.179,A -85,B 0,C 180,E1 -4294.079,E2 -4294.079} C_VEL
LIN {X 0,Y 530.474,Z 672.268,A -85,B 0,C 180,E1 -4295.334,E2 -4295.334} C_VEL
LIN {X 0,Y 530.443,Z 675.488,A -85,B 0,C 180,E1 -4296.579,E2 -4296.579} C_VEL
LIN {X 0,Y 530.411,Z 678.491,A -85,B 0,C 180,E1 -4298.222,E2 -4298.222} C_VEL
LIN {X 0,Y 530.35,Z 680.126,A -85,B 0,C 180,E1 -4299.846,E2 -4299.846} C_VEL
LIN {X 0,Y 530.367,Z 680.409,A -85,B 0,C 180,E1 -4301.456,E2 -4301.456} C_VEL
LIN {X 0,Y 530.365,Z 679.505,A -85,B 0,C 180,E1 -4303.05,E2 -4303.05} C_VEL
LIN {X 0,Y 530.345,Z 677.265,A -85,B 0,C 180,E1 -4304.631,E2 -4304.631} C_VEL
LIN {X 0,Y 530.461,Z 673.853,A -85,B 0,C 180,E1 -4306.203,E2 -4306.203} C_VEL
LIN {X 0,Y 530.527,Z 669.034,A -85,B 0,C 180,E1 -4307.763,E2 -4307.763} C_VEL
LIN {X 0,Y 530.618,Z 662.892,A -85,B 0,C 180,E1 -4309.314,E2 -4309.314} C_VEL
LIN {X 0,Y 530.792,Z 656.216,A -85,B 0,C 180,E1 -4310.665,E2 -4310.665} C_VEL
LIN {X 0,Y 531.033,Z 648.241,A -85,B 0,C 180,E1 -4312.012,E2 -4312.012} C_VEL
LIN {X 0,Y 531.246,Z 638.742,A -85,B 0,C 180,E1 -4313.353,E2 -4313.353} C_VEL
LIN {X 0,Y 531.617,Z 629.039,A -85,B 0,C 180,E1 -4314.5,E2 -4314.5} C_VEL
LIN {X 0,Y 531.979,Z 617.669,A -85,B 0,C 180,E1 -4315.643,E2 -4315.643} C_VEL
LIN {X 0,Y 532.46,Z 603.807,A -85,B 0,C 180,E1 -4316.784,E2 -4316.784} C_VEL
LIN {X 0,Y 532.905,Z 591.179,A -85,B 0,C 180,E1 -4317.638,E2 -4317.638} C_VEL
LIN {X 0,Y 533.297,Z 577.41,A -85,B 0,C 180,E1 -4318.395,E2 -4318.395} C_VEL
LIN {X 0,Y 533.656,Z 563.263,A -85,B 0,C 180,E1 -4319.009,E2 -4319.009} C_VEL
LIN {X 0,Y 534.007,Z 547.028,A -85,B 0,C 180,E1 -4319.529,E2 -4319.529} C_VEL
LIN {X 0,Y 534.222,Z 531.426,A -85,B 0,C 180,E1 -4319.858,E2 -4319.858} C_VEL
LIN {X 0,Y 535.183,Z 382.739,A -85,B 0,C 180,E1 -4321.946,E2 -4321.946} C_VEL
LIN {X 0,Y 532.592,Z 370.767,A -85,B 0,C 180,E1 -4322.239,E2 -4322.239} C_VEL
LIN {X 0,Y 532.907,Z 358.135,A -85,B 0,C 180,E1 -4324.159,E2 -4324.159} C_VEL
LIN {X 0,Y 531.074,Z 348.959,A -85,B 0,C 180,E1 -4325.696,E2 -4325.696} C_VEL
LIN {X 0,Y 531.038,Z 348.965,A -85,B 0,C 180,E1 -4328.371,E2 -4328.371} C_VEL
LIN {X 0,Y 531.054,Z 348.956,A -85,B 0,C 180,E1 -4331.67,E2 -4331.67} C_VEL
LIN {X 0,Y 531.036,Z 348.962,A -85,B 0,C 180,E1 -4334.955,E2 -4334.955} C_VEL
LIN {X 0,Y 530.984,Z 348.967,A -85,B 0,C 180,E1 -4337.723,E2 -4337.723} C_VEL
LIN {X 0,Y 531.029,Z 348.965,A -85,B 0,C 180,E1 -4340.127,E2 -4340.127} C_VEL
LIN {X 0,Y 530.947,Z 348.975,A -85,B 0,C 180,E1 -4342.573,E2 -4342.573} C_VEL
LIN {X 0,Y 530.952,Z 348.969,A -85,B 0,C 180,E1 -4345.06,E2 -4345.06} C_VEL
LIN {X 0,Y 530.954,Z 348.969,A -85,B 0,C 180,E1 -4347.599,E2 -4347.599} C_VEL
LIN {X 0,Y 530.959,Z 348.97,A -85,B 0,C 180,E1 -4350.641,E2 -4350.641} C_VEL
LIN {X 0,Y 530.953,Z 348.971,A -85,B 0,C 180,E1 -4353.775,E2 -4353.775} C_VEL
LIN {X 0,Y 530.906,Z 348.977,A -85,B 0,C 180,E1 -4356.562,E2 -4356.562} C_VEL
LIN {X 0,Y 530.956,Z 348.968,A -85,B 0,C 180,E1 -4359.446,E2 -4359.446} C_VEL
LIN {X 0,Y 530.906,Z 348.977,A -85,B 0,C 180,E1 -4362.464,E2 -4362.464} C_VEL
LIN {X 0,Y 530.96,Z 348.968,A -85,B 0,C 180,E1 -4365.449,E2 -4365.449} C_VEL
LIN {X 0,Y 530.909,Z 348.975,A -85,B 0,C 180,E1 -4368.555,E2 -4368.555} C_VEL
LIN {X 0,Y 530.931,Z 348.975,A -85,B 0,C 180,E1 -4371.526,E2 -4371.526} C_VEL
LIN {X 0,Y 530.927,Z 348.976,A -85,B 0,C 180,E1 -4374.377,E2 -4374.377} C_VEL
LIN {X 0,Y 530.947,Z 348.974,A -85,B 0,C 180,E1 -4377.131,E2 -4377.131} C_VEL
LIN {X 0,Y 530.946,Z 348.979,A -85,B 0,C 180,E1 -4379.801,E2 -4379.801} C_VEL
LIN {X 0,Y 530.952,Z 349.041,A -85,B 0,C 180,E1 -4382.266,E2 -4382.266} C_VEL
LIN {X 0,Y 533.574,Z 360.569,A -85,B 0,C 180,E1 -4383.945,E2 -4383.945} C_VEL
LIN {X 0,Y 533.173,Z 378.593,A -85,B 0,C 180,E1 -4386.294,E2 -4386.294} C_VEL
LIN {X 0,Y 532.62,Z 398.21,A -85,B 0,C 180,E1 -4388.804,E2 -4388.804} C_VEL
LIN {X 0,Y 535.135,Z 411.324,A -85,B 0,C 180,E1 -4389.103,E2 -4389.103} C_VEL
LIN {X 0,Y 534.178,Z 565.158,A -85,B 0,C 180,E1 -4391.258,E2 -4391.258} C_VEL
LIN {X 0,Y 533.893,Z 580.735,A -85,B 0,C 180,E1 -4391.632,E2 -4391.632} C_VEL
LIN {X 0,Y 533.554,Z 596.087,A -85,B 0,C 180,E1 -4392.166,E2 -4392.166} C_VEL
LIN {X 0,Y 533.198,Z 610.834,A -85,B 0,C 180,E1 -4392.846,E2 -4392.846} C_VEL
LIN {X 0,Y 532.738,Z 624.241,A -85,B 0,C 180,E1 -4393.62,E2 -4393.62} C_VEL
LIN {X 0,Y 532.295,Z 637.994,A -85,B 0,C 180,E1 -4394.601,E2 -4394.601} C_VEL
LIN {X 0,Y 531.878,Z 650.23,A -85,B 0,C 180,E1 -4395.654,E2 -4395.654} C_VEL
LIN {X 0,Y 531.565,Z 661.496,A -85,B 0,C 180,E1 -4396.816,E2 -4396.816} C_VEL
LIN {X 0,Y 531.154,Z 672.265,A -85,B 0,C 180,E1 -4398.159,E2 -4398.159} C_VEL
LIN {X 0,Y 530.98,Z 681.29,A -85,B 0,C 180,E1 -4399.513,E2 -4399.513} C_VEL
LIN {X 0,Y 530.76,Z 688.744,A -85,B 0,C 180,E1 -4400.856,E2 -4400.856} C_VEL
LIN {X 0,Y 530.602,Z 695.695,A -85,B 0,C 180,E1 -4402.388,E2 -4402.388} C_VEL
LIN {X 0,Y 530.525,Z 701.159,A -85,B 0,C 180,E1 -4403.915,E2 -4403.915} C_VEL
LIN {X 0,Y 530.413,Z 705.288,A -85,B 0,C 180,E1 -4405.439,E2 -4405.439} C_VEL
LIN {X 0,Y 530.448,Z 708.182,A -85,B 0,C 180,E1 -4406.961,E2 -4406.961} C_VEL
LIN {X 0,Y 530.358,Z 709.908,A -85,B 0,C 180,E1 -4408.48,E2 -4408.48} C_VEL
LIN {X 0,Y 530.339,Z 710.5,A -85,B 0,C 180,E1 -4409.999,E2 -4409.999} C_VEL
LIN {X 0,Y 530.358,Z 709.908,A -85,B 0,C 180,E1 -4411.518,E2 -4411.518} C_VEL
LIN {X 0,Y 530.448,Z 708.181,A -85,B 0,C 180,E1 -4413.037,E2 -4413.037} C_VEL
LIN {X 0,Y 530.412,Z 705.291,A -85,B 0,C 180,E1 -4414.559,E2 -4414.559} C_VEL
LIN {X 0,Y 530.532,Z 701.169,A -85,B 0,C 180,E1 -4416.082,E2 -4416.082} C_VEL
LIN {X 0,Y 530.599,Z 695.706,A -85,B 0,C 180,E1 -4417.61,E2 -4417.61} C_VEL
LIN {X 0,Y 530.758,Z 688.75,A -85,B 0,C 180,E1 -4419.142,E2 -4419.142} C_VEL
LIN {X 0,Y 530.999,Z 680.088,A -85,B 0,C 180,E1 -4420.677,E2 -4420.677} C_VEL
LIN {X 0,Y 531.227,Z 670.692,A -85,B 0,C 180,E1 -4422.05,E2 -4422.05} C_VEL
LIN {X 0,Y 531.562,Z 661.515,A -85,B 0,C 180,E1 -4423.182,E2 -4423.182} C_VEL
LIN {X 0,Y 531.922,Z 649.25,A -85,B 0,C 180,E1 -4424.44,E2 -4424.44} C_VEL
LIN {X 0,Y 532.363,Z 636.997,A -85,B 0,C 180,E1 -4425.483,E2 -4425.483} C_VEL
LIN {X 0,Y 532.738,Z 624.384,A -85,B 0,C 180,E1 -4426.377,E2 -4426.377} C_VEL
LIN {X 0,Y 533.21,Z 611.039,A -85,B 0,C 180,E1 -4427.151,E2 -4427.151} C_VEL
LIN {X 0,Y 533.514,Z 597.538,A -85,B 0,C 180,E1 -4427.784,E2 -4427.784} C_VEL
LIN {X 0,Y 533.866,Z 582.727,A -85,B 0,C 180,E1 -4428.317,E2 -4428.317} C_VEL
LIN {X 0,Y 534.144,Z 567.758,A -85,B 0,C 180,E1 -4428.699,E2 -4428.699} C_VEL
LIN {X 0,Y 534.361,Z 540.422,A -85,B 0,C 180,E1 -4429.125,E2 -4429.125} C_VEL
LIN {X 0,Y 535.072,Z 410.787,A -85,B 0,C 180,E1 -4430.909,E2 -4430.909} C_VEL
LIN {X 0,Y 532.657,Z 398.498,A -85,B 0,C 180,E1 -4431.198,E2 -4431.198} C_VEL
LIN {X 0,Y 533.279,Z 377.494,A -85,B 0,C 180,E1 -4433.905,E2 -4433.905} C_VEL
LIN {X 0,Y 533.724,Z 361.041,A -85,B 0,C 180,E1 -4436.057,E2 -4436.057} C_VEL
LIN {X 0,Y 530.956,Z 348.976,A -85,B 0,C 180,E1 -4437.849,E2 -4437.849} C_VEL
LIN {X 0,Y 530.959,Z 348.973,A -85,B 0,C 180,E1 -4440.642,E2 -4440.642} C_VEL
LIN {X 0,Y 530.954,Z 348.969,A -85,B 0,C 180,E1 -4443.498,E2 -4443.498} C_VEL
LIN {X 0,Y 530.924,Z 348.979,A -85,B 0,C 180,E1 -4446.15,E2 -4446.15} C_VEL
LIN {X 0,Y 530.951,Z 348.971,A -85,B 0,C 180,E1 -4448.652,E2 -4448.652} C_VEL
LIN {X 0,Y 530.952,Z 348.967,A -85,B 0,C 180,E1 -4451.437,E2 -4451.437} C_VEL
LIN {X 0,Y 530.954,Z 348.97,A -85,B 0,C 180,E1 -4454.548,E2 -4454.548} C_VEL
LIN {X 0,Y 530.906,Z 348.974,A -85,B 0,C 180,E1 -4457.536,E2 -4457.536} C_VEL
LIN {X 0,Y 530.955,Z 348.97,A -85,B 0,C 180,E1 -4460.554,E2 -4460.554} C_VEL
LIN {X 0,Y 530.902,Z 348.974,A -85,B 0,C 180,E1 -4463.437,E2 -4463.437} C_VEL
LIN {X 0,Y 530.965,Z 348.969,A -85,B 0,C 180,E1 -4466.497,E2 -4466.497} C_VEL
LIN {X 0,Y 530.947,Z 348.968,A -85,B 0,C 180,E1 -4469.357,E2 -4469.357} C_VEL
LIN {X 0,Y 530.94,Z 348.973,A -85,B 0,C 180,E1 -4472.4,E2 -4472.4} C_VEL
LIN {X 0,Y 530.934,Z 348.969,A -85,B 0,C 180,E1 -4474.939,E2 -4474.939} C_VEL
LIN {X 0,Y 530.96,Z 348.972,A -85,B 0,C 180,E1 -4477.898,E2 -4477.898} C_VEL
LIN {X 0,Y 530.964,Z 348.967,A -85,B 0,C 180,E1 -4480.676,E2 -4480.676} C_VEL
LIN {X 0,Y 530.92,Z 348.971,A -85,B 0,C 180,E1 -4483.069,E2 -4483.069} C_VEL
LIN {X 0,Y 530.991,Z 348.963,A -85,B 0,C 180,E1 -4485.435,E2 -4485.435} C_VEL
LIN {X 0,Y 531.018,Z 348.961,A -85,B 0,C 180,E1 -4488.55,E2 -4488.55} C_VEL
LIN {X 0,Y 530.981,Z 348.966,A -85,B 0,C 180,E1 -4491.628,E2 -4491.628} C_VEL
LIN {X 0,Y 531.074,Z 348.953,A -85,B 0,C 180,E1 -4494.685,E2 -4494.685} C_VEL
LIN {X 0,Y 531.119,Z 348.951,A -85,B 0,C 180,E1 -4497.725,E2 -4497.725} C_VEL
LIN {X 0,Y 531.113,Z 348.957,A -85,B 0,C 180,E1 -4500,E2 -4500} C_VEL
LIN {X 0,Y 531.118,Z 348.951,A -85,B 0,C 180,E1 -4502.275,E2 -4502.275} C_VEL
LIN {X 0,Y 531.068,Z 348.953,A -85,B 0,C 180,E1 -4505.315,E2 -4505.315} C_VEL
LIN {X 0,Y 530.973,Z 348.968,A -85,B 0,C 180,E1 -4508.372,E2 -4508.372} C_VEL
LIN {X 0,Y 530.996,Z 348.966,A -85,B 0,C 180,E1 -4511.651,E2 -4511.651} C_VEL
LIN {X 0,Y 531.008,Z 348.96,A -85,B 0,C 180,E1 -4514.953,E2 -4514.953} C_VEL
LIN {X 0,Y 530.951,Z 348.969,A -85,B 0,C 180,E1 -4518.523,E2 -4518.523} C_VEL
LIN {X 0,Y 530.976,Z 348.964,A -85,B 0,C 180,E1 -4520.939,E2 -4520.939} C_VEL
LIN {X 0,Y 530.939,Z 348.976,A -85,B 0,C 180,E1 -4524.032,E2 -4524.032} C_VEL
LIN {X 0,Y 530.931,Z 348.97,A -85,B 0,C 180,E1 -4526.748,E2 -4526.748} C_VEL
LIN {X 0,Y 530.947,Z 348.969,A -85,B 0,C 180,E1 -4529.325,E2 -4529.325} C_VEL
LIN {X 0,Y 530.952,Z 348.973,A -85,B 0,C 180,E1 -4532.101,E2 -4532.101} C_VEL
LIN {X 0,Y 530.947,Z 348.967,A -85,B 0,C 180,E1 -4534.85,E2 -4534.85} C_VEL
LIN {X 0,Y 530.921,Z 348.975,A -85,B 0,C 180,E1 -4537.512,E2 -4537.512} C_VEL
LIN {X 0,Y 530.937,Z 348.97,A -85,B 0,C 180,E1 -4540.437,E2 -4540.437} C_VEL
LIN {X 0,Y 530.916,Z 348.975,A -85,B 0,C 180,E1 -4543.532,E2 -4543.532} C_VEL
LIN {X 0,Y 530.251,Z 349.059,A -85,B 0,C 180,E1 -4544.166,E2 -4544.166} C_VEL
LIN {X 0,Y 527.414,Z 349.409,A -85,B 0,C 180,E1 -4545.195,E2 -4545.195} C_VEL
LIN {X 0,Y 525.01,Z 349.713,A -85,B 0,C 180,E1 -4546.023,E2 -4546.023} C_VEL
LIN {X 0,Y 523.968,Z 349.838,A -85,B 0,C 180,E1 -4546.663,E2 -4546.663} C_VEL
LIN {X 0,Y 523.878,Z 349.848,A -85,B 0,C 180,E1 -4546.88,E2 -4546.88} C_VEL
LIN {X 0,Y 523.905,Z 349.852,A -85,B 0,C 180,E1 -4549.919,E2 -4549.919} C_VEL
LIN {X 0,Y 523.876,Z 349.848,A -85,B 0,C 180,E1 -4552.867,E2 -4552.867} C_VEL
LIN {X 0,Y 523.912,Z 349.852,A -85,B 0,C 180,E1 -4555.71,E2 -4555.71} C_VEL
LIN {X 0,Y 523.913,Z 349.845,A -85,B 0,C 180,E1 -4558.457,E2 -4558.457} C_VEL
LIN {X 0,Y 523.894,Z 349.847,A -85,B 0,C 180,E1 -4561.124,E2 -4561.124} C_VEL
LIN {X 0,Y 523.906,Z 349.85,A -85,B 0,C 180,E1 -4563.999,E2 -4563.999} C_VEL
LIN {X 0,Y 523.906,Z 349.847,A -85,B 0,C 180,E1 -4566.271,E2 -4566.271} C_VEL
LIN {X 0,Y 523.943,Z 349.84,A -85,B 0,C 180,E1 -4568.768,E2 -4568.768} C_VEL
LIN {X 0,Y 523.934,Z 349.843,A -85,B 0,C 180,E1 -4571.222,E2 -4571.222} C_VEL
LIN {X 0,Y 523.903,Z 349.853,A -85,B 0,C 180,E1 -4573.639,E2 -4573.639} C_VEL
LIN {X 0,Y 523.925,Z 349.847,A -85,B 0,C 180,E1 -4576.029,E2 -4576.029} C_VEL
LIN {X 0,Y 524.015,Z 349.832,A -85,B 0,C 180,E1 -4578.395,E2 -4578.395} C_VEL
LIN {X 0,Y 523.956,Z 349.845,A -85,B 0,C 180,E1 -4581.516,E2 -4581.516} C_VEL
LIN {X 0,Y 524.036,Z 349.828,A -85,B 0,C 180,E1 -4584.614,E2 -4584.614} C_VEL
LIN {X 0,Y 524.108,Z 349.829,A -85,B 0,C 180,E1 -4587.696,E2 -4587.696} C_VEL
LIN {X 0,Y 524.1,Z 349.824,A -85,B 0,C 180,E1 -4590.001,E2 -4590.001} C_VEL
LIN {X 0,Y 524.108,Z 349.82,A -85,B 0,C 180,E1 -4592.307,E2 -4592.307} C_VEL
LIN {X 0,Y 524.013,Z 349.833,A -85,B 0,C 180,E1 -4596.16,E2 -4596.16} C_VEL
LIN {X 0,Y 523.984,Z 349.839,A -85,B 0,C 180,E1 -4599.263,E2 -4599.263} C_VEL
LIN {X 0,Y 524.003,Z 349.84,A -85,B 0,C 180,E1 -4601.737,E2 -4601.737} C_VEL
LIN {X 0,Y 523.997,Z 349.835,A -85,B 0,C 180,E1 -4605.052,E2 -4605.052} C_VEL
LIN {X 0,Y 523.92,Z 349.846,A -85,B 0,C 180,E1 -4607.972,E2 -4607.972} C_VEL
LIN {X 0,Y 523.964,Z 349.838,A -85,B 0,C 180,E1 -4610.411,E2 -4610.411} C_VEL
LIN {X 0,Y 523.913,Z 349.845,A -85,B 0,C 180,E1 -4612.894,E2 -4612.894} C_VEL
LIN {X 0,Y 523.906,Z 349.852,A -85,B 0,C 180,E1 -4615.422,E2 -4615.422} C_VEL
LIN {X 0,Y 523.916,Z 349.846,A -85,B 0,C 180,E1 -4618.003,E2 -4618.003} C_VEL
LIN {X 0,Y 523.942,Z 349.841,A -85,B 0,C 180,E1 -4620.853,E2 -4620.853} C_VEL
LIN {X 0,Y 523.951,Z 349.845,A -85,B 0,C 180,E1 -4623.732,E2 -4623.732} C_VEL
LIN {X 0,Y 523.903,Z 349.847,A -85,B 0,C 180,E1 -4626.401,E2 -4626.401} C_VEL
LIN {X 0,Y 523.924,Z 349.847,A -85,B 0,C 180,E1 -4629.085,E2 -4629.085} C_VEL
LIN {X 0,Y 523.946,Z 349.844,A -85,B 0,C 180,E1 -4632.12,E2 -4632.12} C_VEL
LIN {X 0,Y 523.943,Z 349.849,A -85,B 0,C 180,E1 -4635.311,E2 -4635.311} C_VEL
LIN {X 0,Y 523.969,Z 349.987,A -85,B 0,C 180,E1 -4636.278,E2 -4636.278} C_VEL
LIN {X 0,Y 525.876,Z 359.245,A -85,B 0,C 180,E1 -4637.821,E2 -4637.821} C_VEL
LIN {X 0,Y 525.664,Z 370.797,A -85,B 0,C 180,E1 -4639.566,E2 -4639.566} C_VEL
LIN {X 0,Y 528.51,Z 384.13,A -85,B 0,C 180,E1 -4639.89,E2 -4639.89} C_VEL
LIN {X 0,Y 527.451,Z 535.869,A -85,B 0,C 180,E1 -4642.063,E2 -4642.063} C_VEL
LIN {X 0,Y 527.17,Z 551.586,A -85,B 0,C 180,E1 -4642.446,E2 -4642.446} C_VEL
LIN {X 0,Y 526.8,Z 566.789,A -85,B 0,C 180,E1 -4642.986,E2 -4642.986} C_VEL
LIN {X 0,Y 526.365,Z 580.085,A -85,B 0,C 180,E1 -4643.606,E2 -4643.606} C_VEL
LIN {X 0,Y 525.951,Z 593.06,A -85,B 0,C 180,E1 -4644.357,E2 -4644.357} C_VEL
LIN {X 0,Y 525.51,Z 605.758,A -85,B 0,C 180,E1 -4645.246,E2 -4645.246} C_VEL
LIN {X 0,Y 525.052,Z 618.254,A -85,B 0,C 180,E1 -4646.305,E2 -4646.305} C_VEL
LIN {X 0,Y 524.655,Z 628.959,A -85,B 0,C 180,E1 -4647.396,E2 -4647.396} C_VEL
LIN {X 0,Y 524.306,Z 639.461,A -85,B 0,C 180,E1 -4648.659,E2 -4648.659} C_VEL
LIN {X 0,Y 523.979,Z 648.952,A -85,B 0,C 180,E1 -4650.024,E2 -4650.024} C_VEL
LIN {X 0,Y 523.741,Z 656.479,A -85,B 0,C 180,E1 -4651.332,E2 -4651.332} C_VEL
LIN {X 0,Y 523.572,Z 663.752,A -85,B 0,C 180,E1 -4652.845,E2 -4652.845} C_VEL
LIN {X 0,Y 523.465,Z 668.582,A -85,B 0,C 180,E1 -4654.098,E2 -4654.098} C_VEL
LIN {X 0,Y 523.377,Z 672.674,A -85,B 0,C 180,E1 -4655.4,E2 -4655.4} C_VEL
LIN {X 0,Y 523.303,Z 676.664,A -85,B 0,C 180,E1 -4657.078,E2 -4657.078} C_VEL
LIN {X 0,Y 523.293,Z 678.154,A -85,B 0,C 180,E1 -4657.926,E2 -4657.926} C_VEL
LIN {X 0,Y 523.257,Z 679.917,A -85,B 0,C 180,E1 -4659.561,E2 -4659.561} C_VEL
LIN {X 0,Y 523.261,Z 680.473,A -85,B 0,C 180,E1 -4661.195,E2 -4661.195} C_VEL
LIN {X 0,Y 523.292,Z 679.704,A -85,B 0,C 180,E1 -4662.814,E2 -4662.814} C_VEL
LIN {X 0,Y 523.245,Z 677.73,A -85,B 0,C 180,E1 -4664.417,E2 -4664.417} C_VEL
LIN {X 0,Y 523.312,Z 676.269,A -85,B 0,C 180,E1 -4665.23,E2 -4665.23} C_VEL
LIN {X 0,Y 523.368,Z 672.348,A -85,B 0,C 180,E1 -4666.804,E2 -4666.804} C_VEL
LIN {X 0,Y 523.459,Z 667.195,A -85,B 0,C 180,E1 -4668.381,E2 -4668.381} C_VEL
LIN {X 0,Y 523.633,Z 660.552,A -85,B 0,C 180,E1 -4669.951,E2 -4669.951} C_VEL
LIN {X 0,Y 523.823,Z 653.43,A -85,B 0,C 180,E1 -4671.318,E2 -4671.318} C_VEL
LIN {X 0,Y 524.113,Z 644.909,A -85,B 0,C 180,E1 -4672.681,E2 -4672.681} C_VEL
LIN {X 0,Y 524.437,Z 634.648,A -85,B 0,C 180,E1 -4674.038,E2 -4674.038} C_VEL
LIN {X 0,Y 524.819,Z 624.252,A -85,B 0,C 180,E1 -4675.199,E2 -4675.199} C_VEL
LIN {X 0,Y 525.22,Z 612.865,A -85,B 0,C 180,E1 -4676.26,E2 -4676.26} C_VEL
LIN {X 0,Y 525.706,Z 600.645,A -85,B 0,C 180,E1 -4677.222,E2 -4677.222} C_VEL
LIN {X 0,Y 526.172,Z 587.295,A -85,B 0,C 180,E1 -4678.086,E2 -4678.086} C_VEL
LIN {X 0,Y 526.621,Z 572.419,A -85,B 0,C 180,E1 -4678.853,E2 -4678.853} C_VEL
LIN {X 0,Y 526.975,Z 557.373,A -85,B 0,C 180,E1 -4679.446,E2 -4679.446} C_VEL
LIN {X 0,Y 527.324,Z 542.131,A -85,B 0,C 180,E1 -4679.88,E2 -4679.88} C_VEL
LIN {X 0,Y 527.473,Z 525.765,A -85,B 0,C 180,E1 -4680.176,E2 -4680.176} C_VEL
LIN {X 0,Y 528.527,Z 383.637,A -85,B 0,C 180,E1 -4682.21,E2 -4682.21} C_VEL
LIN {X 0,Y 525.759,Z 370.994,A -85,B 0,C 180,E1 -4682.535,E2 -4682.535} C_VEL
LIN {X 0,Y 526.063,Z 360.099,A -85,B 0,C 180,E1 -4684.214,E2 -4684.214} C_VEL
LIN {X 0,Y 524.509,Z 352.012,A -85,B 0,C 180,E1 -4685.575,E2 -4685.575} C_VEL
LIN {X 0,Y 524.05,Z 349.835,A -85,B 0,C 180,E1 -4685.966,E2 -4685.966} C_VEL
LIN {X 0,Y 523.99,Z 349.844,A -85,B 0,C 180,E1 -4688.484,E2 -4688.484} C_VEL
LIN {X 0,Y 524.004,Z 349.835,A -85,B 0,C 180,E1 -4691.737,E2 -4691.737} C_VEL
LIN {X 0,Y 523.998,Z 349.838,A -85,B 0,C 180,E1 -4695.052,E2 -4695.052} C_VEL
LIN {X 0,Y 523.948,Z 349.845,A -85,B 0,C 180,E1 -4697.969,E2 -4697.969} C_VEL
LIN {X 0,Y 523.976,Z 349.845,A -85,B 0,C 180,E1 -4700.41,E2 -4700.41} C_VEL
LIN {X 0,Y 523.912,Z 349.848,A -85,B 0,C 180,E1 -4702.893,E2 -4702.893} C_VEL
LIN {X 0,Y 523.901,Z 349.847,A -85,B 0,C 180,E1 -4705.421,E2 -4705.421} C_VEL
LIN {X 0,Y 523.899,Z 349.852,A -85,B 0,C 180,E1 -4708.003,E2 -4708.003} C_VEL
LIN {X 0,Y 523.911,Z 349.846,A -85,B 0,C 180,E1 -4710.847,E2 -4710.847} C_VEL
LIN {X 0,Y 523.929,Z 349.846,A -85,B 0,C 180,E1 -4713.728,E2 -4713.728} C_VEL
LIN {X 0,Y 523.86,Z 349.857,A -85,B 0,C 180,E1 -4716.394,E2 -4716.394} C_VEL
LIN {X 0,Y 523.906,Z 349.846,A -85,B 0,C 180,E1 -4719.086,E2 -4719.086} C_VEL
LIN {X 0,Y 523.888,Z 349.855,A -85,B 0,C 180,E1 -4722.125,E2 -4722.125} C_VEL
LIN {X 0,Y 523.931,Z 349.843,A -85,B 0,C 180,E1 -4725.311,E2 -4725.311} C_VEL
LIN {X 0,Y 523.877,Z 349.85,A -85,B 0,C 180,E1 -4728.699,E2 -4728.699} C_VEL
LIN {X 0,Y 523.89,Z 349.856,A -85,B 0,C 180,E1 -4731.895,E2 -4731.895} C_VEL
LIN {X 0,Y 523.89,Z 349.85,A -85,B 0,C 180,E1 -4734.916,E2 -4734.916} C_VEL
LIN {X 0,Y 523.901,Z 349.856,A -85,B 0,C 180,E1 -4737.686,E2 -4737.686} C_VEL
LIN {X 0,Y 523.937,Z 349.848,A -85,B 0,C 180,E1 -4740.68,E2 -4740.68} C_VEL
LIN {X 0,Y 523.935,Z 350.043,A -85,B 0,C 180,E1 -4742.025,E2 -4742.025} C_VEL
LIN {X 0,Y 526.764,Z 362.53,A -85,B 0,C 180,E1 -4743.877,E2 -4743.877} C_VEL
LIN {X 0,Y 526.186,Z 383.22,A -85,B 0,C 180,E1 -4746.607,E2 -4746.607} C_VEL
LIN {X 0,Y 525.745,Z 398.196,A -85,B 0,C 180,E1 -4748.519,E2 -4748.519} C_VEL
LIN {X 0,Y 528.464,Z 412.705,A -85,B 0,C 180,E1 -4748.855,E2 -4748.855} C_VEL
LIN {X 0,Y 527.393,Z 565.115,A -85,B 0,C 180,E1 -4751.035,E2 -4751.035} C_VEL
LIN {X 0,Y 527.086,Z 580.527,A -85,B 0,C 180,E1 -4751.411,E2 -4751.411} C_VEL
LIN {X 0,Y 526.722,Z 595.286,A -85,B 0,C 180,E1 -4751.926,E2 -4751.926} C_VEL
LIN {X 0,Y 526.302,Z 610.157,A -85,B 0,C 180,E1 -4752.614,E2 -4752.614} C_VEL
LIN {X 0,Y 525.85,Z 623.644,A -85,B 0,C 180,E1 -4753.4,E2 -4753.4} C_VEL
LIN {X 0,Y 525.411,Z 637.356,A -85,B 0,C 180,E1 -4754.383,E2 -4754.383} C_VEL
LIN {X 0,Y 524.926,Z 649.774,A -85,B 0,C 180,E1 -4755.46,E2 -4755.46} C_VEL
LIN {X 0,Y 524.545,Z 661.094,A -85,B 0,C 180,E1 -4756.636,E2 -4756.636} C_VEL
LIN {X 0,Y 524.139,Z 672.063,A -85,B 0,C 180,E1 -4758.004,E2 -4758.004} C_VEL
LIN {X 0,Y 523.925,Z 681.175,A -85,B 0,C 180,E1 -4759.37,E2 -4759.37} C_VEL
LIN {X 0,Y 523.7,Z 688.718,A -85,B 0,C 180,E1 -4760.732,E2 -4760.732} C_VEL
LIN {X 0,Y 523.536,Z 695.695,A -85,B 0,C 180,E1 -4762.284,E2 -4762.284} C_VEL
LIN {X 0,Y 523.438,Z 701.158,A -85,B 0,C 180,E1 -4763.833,E2 -4763.833} C_VEL
LIN {X 0,Y 523.324,Z 705.287,A -85,B 0,C 180,E1 -4765.377,E2 -4765.377} C_VEL
LIN {X 0,Y 523.358,Z 708.182,A -85,B 0,C 180,E1 -4766.92,E2 -4766.92} C_VEL
LIN {X 0,Y 523.272,Z 709.908,A -85,B 0,C 180,E1 -4768.46,E2 -4768.46} C_VEL
LIN {X 0,Y 523.243,Z 710.5,A -85,B 0,C 180,E1 -4769.999,E2 -4769.999} C_VEL
LIN {X 0,Y 523.271,Z 709.907,A -85,B 0,C 180,E1 -4771.538,E2 -4771.538} C_VEL
LIN {X 0,Y 523.357,Z 708.18,A -85,B 0,C 180,E1 -4773.078,E2 -4773.078} C_VEL
LIN {X 0,Y 523.323,Z 705.29,A -85,B 0,C 180,E1 -4774.621,E2 -4774.621} C_VEL
LIN {X 0,Y 523.449,Z 701.169,A -85,B 0,C 180,E1 -4776.165,E2 -4776.165} C_VEL
